// Return if no parameter is remaining...
IF ( ParameterCnt = 0 ) THEN RETURN; END_IF
// dec remaining parameter(s)                        
ParameterCnt := ParameterCnt - 1;
// Create log entry for OriginID
CreateLogMessagePara1 ( Timestamp   := Timestamp,
                        MessageType := MessageType.CMD,
                        Severity    := Severity.DEBUG,
                        MessageCode := 0,
                        MessageText := 'Response.OriginID = {1}',
                        Para1       :=  INT_TO_STRING(_response.OriginID));                       
                
END_METHOD

METHOD PROTECTED Reset : DINT
VAR_INPUT
END_VAR
                  Reset := SUPER^.Reset();

Done               := FALSE;
Busy               := FALSE;
ParameterAccepted  := FALSE;
CommandBuffered    := FALSE;
CommandAborted     := FALSE;
CommandInterrupted := FALSE;

                
END_METHOD
END_FUNCTION_BLOCK

/// Write default values of dynamic parameters used by move commands
FUNCTION_BLOCK MC_WriteRobotDefaultDynamicsFB EXTENDS RobotLibraryBaseExecuteFB
// ------------------------------------------------------------------------- 
//  SRCI Robot Library                                                
// ------------------------------------------------------------------------- 
//                                                                           
//  Object:      WriteRobotDefaultDynamicsFB                                       
//  Author:      Thorsten Brach                                                
//  Date:        2024-06-01
//
//  Description:                                              
//   
//                                                                           
//  Copyright: 
//    (C) 2024 Thorsten Brach. All rights reserved                                                                                                                                            
//             Licensed under the MIT License.
//                                                                           
//  Disclaimer:                                                                           
//    This project is provided without any guarantee and can be used for   
//    private and commercial purposes. Any use is at the user’s 
//    own risk and responsibility.
//
// -------------------------------------------------------------------------
VAR_INPUT
  /// command parameter 
  ParCmd             : WriteRobotDefaultDynamicsParCmd;
END_VAR
VAR_OUTPUT
  /// Command is transferred and confirmed by the RC
  CommandBuffered    : BOOL;
  /// The command was aborted by another command
  CommandAborted     : BOOL;
  /// TRUE, while command is interrupted during execution and can be continued.
  CommandInterrupted : BOOL;
  /// command outputs
  OutCmd             : WriteRobotDefaultDynamicsOutCmd;       
END_VAR

VAR
  /// internal copy of command parameter 
 _parCmd             : WriteRobotDefaultDynamicsParCmd;
  /// command data to send
 _command            : WriteRobotDefaultDynamicsSendData;
  /// response data received
 _response           : WriteRobotDefaultDynamicsRecvData;      
END_VAR

            SUPER^(AxesGroup := AxesGroup);
          

METHOD INTERNAL CheckAddParameter : BOOL
VAR_INPUT
  /// Payload pointer
  PayloadPtr : UDINT;
END_VAR
VAR
  /// Payload as byte array
  Payload    : ARRAY [1..SIZEOF(_command)] OF BYTE;
  /// Null Byte array 
  Null       : ARRAY [1..SIZEOF(_command)] OF BYTE;
  /// Data length to compare
  DataLen    : UDINT;
END_VAR
                  // Payload pointer must be decreased by one byte, because ADR(Payload) is already one byte !
PayloadPtr := LIMIT (0, PayloadPtr - 1, SIZEOF(Payload) -1);
// Convert command struct to payload array
SysDepMemCpy( pDest := ADR(Payload), pSrc := ADR(_command), DataLen := SIZEOF(_command));
// Calculate the data length to compare - at least one byte must be compared !
DataLen := LIMIT(1, SIZEOF(Payload) - PayloadPtr, SIZEOF(Payload)); 
// Compare Payload-Array with Null-Byte-Array
CheckAddParameter := SysDepMemCmp( pData1 := ADR(Payload) + PayloadPtr , pData2 := ADR(Null), DataLen := DataLen) <>  RobotLibraryConstants.OK ;
                
END_METHOD

METHOD PROTECTED CheckFunctionSupported : BOOL
VAR_IN_OUT
  /// Robot assignment of function
  AxesGroup : AxesGroup; 
END_VAR
                  CheckFunctionSupported := AxesGroup.State.RobotData.RCSupportedFunctions.WriteRobotDefaultDynamics;

IF ( NOT CheckFunctionSupported )
THEN
  // call base implementation for set error and create log entry
  SUPER^.CheckFunctionSupported(AxesGroup := AxesGroup);
END_IF
                
END_METHOD

METHOD PROTECTED CheckParameterChanged : BOOL
VAR_IN_OUT
  /// Robot assignment of function
  AxesGroup    : AxesGroup; 
END_VAR
                  // Check ParCmd Size is > 0, because MemCmp does not work correctly with size = 0
IF (SIZEOF(ParCmd) = 0) OR (_stepCmd = 0)
THEN 
  RETURN;
END_IF

// compare memory 
_parameterChanged := ( SysDepMemCmp(pData1 := ADR(ParCmd), pData2 := ADR(_parCmd), DataLen := SIZEOF(ParCmd)) <> RobotLibraryConstants.OK );

// check parameter valid ?
_parameterValid   := CheckParameterValid( AxesGroup := AxesGroup );

IF ((  _parameterChanged        )  AND 
    (  _parameterValid          )) OR
    (  _parameterUpdateInternal )  
THEN  
  // Create log entry for parameter changed event
  CreateLogMessagePara1 ( Timestamp   := AxesGroup.State.SystemTime,
                          MessageType := MessageType.CMD,
                          Severity    := Severity.DEBUG,
                          MessageCode := 0,
                          MessageText := 'NotifyParameterChanged Event {1}',
                          Para1       :=  '' );

  // reset internal flag for send parameter update
 _parameterUpdateInternal := FALSE;
  // update internal copy of parameters 
 _parCmd := ParCmd;
  // inc parameter sequence
 _command.ParSeq := _command.ParSeq + 1;
  // update command data  
  CommandData := CreateCommandPayload(AxesGroup := AxesGroup); // ( Access via reference to rCommandFB in ACR )
  // notify active command register 
  AxesGroup.Acyclic.ActiveCommandRegister.NotifyParameterChanged := _uniqueID;
END_IF
                
END_METHOD

METHOD PROTECTED CheckParameterValid : BOOL
VAR_IN_OUT
  /// Robot assignment of function
  AxesGroup : AxesGroup; 
END_VAR
VAR
  /// internal index for loops
 _idx : DINT;
END_VAR
                  CheckParameterValid := TRUE;


// Check ParCmd.DynamicValues.VelocityRate ? 
IF ( SysDepIsValidReal(ParCmd.DynamicValues.VelocityRate) = FALSE ) 
THEN
  // Parameter not valid
  CheckParameterValid := FALSE;
  // Set error
  SetError( ErrorID := RobotLibraryErrorIdEnum.ERR_VELOCITY_INVALID, Overwrite := TRUE );
  
  // Create log entry
  CreateLogMessagePara1 ( Timestamp   := AxesGroup.State.SystemTime,
                          MessageType := MessageType.CMD,
                          Severity    := Severity.ERROR,
                          MessageCode := ErrorID,
                          MessageText := 'Invalid Parameter ParCmd.DynamicValues.VelocityRate = {1}',
                          Para1       := VALID_REAL_TO_STRING(ParCmd.DynamicValues.VelocityRate));

  RETURN;                          
END_IF


// Check ParCmd.DynamicValues.AccelerationRate ? 
IF ( SysDepIsValidReal(ParCmd.DynamicValues.AccelerationRate) = FALSE ) 
THEN
  // Parameter not valid
  CheckParameterValid := FALSE;
  // Set error
  SetError( ErrorID := RobotLibraryErrorIdEnum.ERR_ACCELERATION_INVALID, Overwrite := TRUE );
  
  // Create log entry
  CreateLogMessagePara1 ( Timestamp   := AxesGroup.State.SystemTime,
                          MessageType := MessageType.CMD,
                          Severity    := Severity.ERROR,
                          MessageCode := ErrorID,
                          MessageText := 'Invalid Parameter ParCmd.DynamicValues.AccelerationRate = {1}',
                          Para1       := VALID_REAL_TO_STRING(ParCmd.DynamicValues.AccelerationRate));

  RETURN;                          
END_IF


// Check ParCmd.DynamicValues.DecelerationRate ? 
IF ( SysDepIsValidReal(ParCmd.DynamicValues.DecelerationRate) = FALSE ) 
THEN
  // Parameter not valid
  CheckParameterValid := FALSE;
  // Set error
  SetError( ErrorID := RobotLibraryErrorIdEnum.ERR_DECELERATION_INVALID, Overwrite := TRUE );
  
  // Create log entry
  CreateLogMessagePara1 ( Timestamp   := AxesGroup.State.SystemTime,
                          MessageType := MessageType.CMD,
                          Severity    := Severity.ERROR,
                          MessageCode := ErrorID,
                          MessageText := 'Invalid Parameter ParCmd.DynamicValues.DecelerationRate = {1}',
                          Para1       := VALID_REAL_TO_STRING(ParCmd.DynamicValues.DecelerationRate));

  RETURN;                          
END_IF


// Check ParCmd.DynamicValues.JerkRate ? 
IF ( SysDepIsValidReal(ParCmd.DynamicValues.JerkRate) = FALSE ) 
THEN
  // Parameter not valid
  CheckParameterValid := FALSE;
  // Set error
  SetError( ErrorID := RobotLibraryErrorIdEnum.ERR_JERK_INVALID, Overwrite := TRUE );
  
  // Create log entry
  CreateLogMessagePara1 ( Timestamp   := AxesGroup.State.SystemTime,
                          MessageType := MessageType.CMD,
                          Severity    := Severity.ERROR,
                          MessageCode := ErrorID,
                          MessageText := 'Invalid Parameter ParCmd.DynamicValues.JerkRate = {1}',
                          Para1       := VALID_REAL_TO_STRING(ParCmd.DynamicValues.JerkRate));

  RETURN;                          
END_IF
                
END_METHOD

METHOD INTERNAL CreateCommandPayload : RobotLibraryCommandDataFB
VAR_IN_OUT
  /// Robot assignment of function
  AxesGroup : AxesGroup; 
END_VAR
VAR
  /// Parameter count
 _parameterCnt : DINT;
END_VAR
// Table 6-146: Sent CMD payload (PLC to RC) of "WriteRobotDefaultDynamics"
// --------------------------
// Header
// --------------------------
// Byte 00 : UINT  - Type HB     
// Byte 01 :       - Type LB    
// Byte 02 : USINT - Reserve | ExecutionMode
// Byte 03 : USINT - ParSeq  | Priority
// --------------------------
// Datablock
// --------------------------
// Byte 04 : DATE Date
// Byte 05 : 
// Byte 06 : TIME_OF_DAY Time
// Byte 07 : 
// Byte 08 : 
// Byte 09 : UINT VelocityRate
// Byte 10 : 
// Byte 11 : 
// Byte 12 : UINT AccelerationRate
// Byte 13 : 
// Byte 14 : 
// Byte 15 : UINT DecelerationRate
// Byte 16 : 
// Byte 17 : 
// Byte 18 : UINT JerkRate
// --------------------------
                  // set command parameter 
_command.CmdTyp           :=  CmdType.WriteRobotDefaultDynamics;
_command.ExecMode         :=  ExecMode;
_command.ParSeq           := _command.ParSeq;
_command.Priority         :=  Priority;
_command.Timestamp        := _parCmd.DynamicValues.Timestamp;
_command.VelocityRate     := REAL_TO_PERCENT_UINT(_parCmd.DynamicValues.VelocityRate     , IsOptional := FALSE);
_command.AccelerationRate := REAL_TO_PERCENT_UINT(_parCmd.DynamicValues.AccelerationRate , IsOptional := FALSE);
_command.JerkRate         := REAL_TO_PERCENT_UINT(_parCmd.DynamicValues.JerkRate         , IsOptional := TRUE );
_command.DecelerationRate := REAL_TO_PERCENT_UINT(_parCmd.DynamicValues.DecelerationRate , IsOptional := TRUE );

// copy command data to header
_cmdHeader := _command;
// call base implementation to copy header to payload buffer
CreateCommandPayload := SUPER^.CreateCommandPayload(AxesGroup := AxesGroup);


// Check parameter must be added ? 
IF ( CheckAddParameter(CreateCommandPayload.PayloadPtr))
THEN
  // add command.DynamicValues.Timestamp.IEC_DATE
  CreateCommandPayload.AddUint(_command.Timestamp.IEC_DATE);
  // inc parameter counter
 _parameterCnt := _parameterCnt + 1;  
END_IF


// Check parameter must be added ? 
IF ( CheckAddParameter(CreateCommandPayload.PayloadPtr))
THEN
  // add command.DynamicValues.Timestamp.IEC_TIME
  CreateCommandPayload.AddTime(_command.Timestamp.IEC_TIME);
  // inc parameter counter
 _parameterCnt := _parameterCnt + 1;  
END_IF


// Check parameter must be added ? 
IF ( CheckAddParameter(CreateCommandPayload.PayloadPtr))
THEN
  // add command.DynamicValues.VelocityRate
  CreateCommandPayload.AddUint(_command.VelocityRate);
  // inc parameter counter
 _parameterCnt := _parameterCnt + 1;  
END_IF


// Check parameter must be added ? 
IF ( CheckAddParameter(CreateCommandPayload.PayloadPtr))
THEN
  // add command.DynamicValues.AccelerationRate
  CreateCommandPayload.AddUint(_command.AccelerationRate);
  // inc parameter counter
 _parameterCnt := _parameterCnt + 1;  
END_IF


// Check parameter must be added ? 
IF ( CheckAddParameter(CreateCommandPayload.PayloadPtr))
THEN
  // add command.DynamicValues.DecelerationRate
  CreateCommandPayload.AddUint(_command.DecelerationRate);
  // inc parameter counter
 _parameterCnt := _parameterCnt + 1;  
END_IF


// Check parameter must be added ? 
IF ( CheckAddParameter(CreateCommandPayload.PayloadPtr))
THEN
  // add command.DynamicValues.JerkRate
  CreateCommandPayload.AddUint(_command.JerkRate);
  // inc parameter counter
 _parameterCnt := _parameterCnt + 1;  
END_IF

 
// Create logging
CreateCommandPayloadLog(AxesGroup := AxesGroup, ParameterCnt := _parameterCnt);
                
END_METHOD

METHOD INTERNAL CreateCommandPayloadLog
VAR_IN_OUT
  /// Robot assignment of function
  AxesGroup : AxesGroup; 
END_VAR
VAR_INPUT
  /// Parameter count
  ParameterCnt : DINT;
END_VAR
                  // Create log entry for Parameter start
CreateLogMessagePara1 ( Timestamp   := AxesGroup.State.SystemTime,
                        MessageType := MessageType.CMD,
                        Severity    := Severity.DEBUG,
                        MessageCode := 0,
                        MessageText := 'Create command payload with {1} parameter(s) :',
                        Para1       := DINT_TO_STRING(ParameterCnt));
  

// Return if no parameter is remaining...
IF ( ParameterCnt = 0 ) THEN RETURN; END_IF
// dec remaining parameter(s)                        
ParameterCnt := ParameterCnt - 1;
// Create log entry for Timestamp.IEC_DATE
CreateLogMessagePara1 ( Timestamp   := AxesGroup.State.SystemTime,
                        MessageType := MessageType.CMD,
                        Severity    := Severity.DEBUG,
                        MessageCode := 0,
                        MessageText := 'Command.Timestamp.IEC_DATE = {1}',
                        Para1       :=  IEC_DATE_TO_STRING(_command.Timestamp.IEC_DATE));


// Return if no parameter is remaining...
IF ( ParameterCnt = 0 ) THEN RETURN; END_IF
// dec remaining parameter(s)                        
ParameterCnt := ParameterCnt - 1;
// Create log entry for Timestamp.IEC_TIME
CreateLogMessagePara1 ( Timestamp   := AxesGroup.State.SystemTime,
                        MessageType := MessageType.CMD,
                        Severity    := Severity.DEBUG,
                        MessageCode := 0,
                        MessageText := 'Command.Timestamp.IEC_TIME = {1}',
                        Para1       :=  IEC_TIME_TO_STRING(_command.Timestamp.IEC_TIME));


// Return if no parameter is remaining...
IF ( ParameterCnt = 0 ) THEN RETURN; END_IF
// dec remaining parameter(s)                        
ParameterCnt := ParameterCnt - 1;
// Create log entry for VelocityRate
CreateLogMessagePara1 ( Timestamp   := AxesGroup.State.SystemTime,
                        MessageType := MessageType.CMD,
                        Severity    := Severity.DEBUG,
                        MessageCode := 0,
                        MessageText := 'Command.VelocityRate = {1}',
                        Para1       :=  UINT_TO_STRING(_command.VelocityRate));


// Return if no parameter is remaining...
IF ( ParameterCnt = 0 ) THEN RETURN; END_IF
// dec remaining parameter(s)                        
ParameterCnt := ParameterCnt - 1;
// Create log entry for AccelerationRate
CreateLogMessagePara1 ( Timestamp   := AxesGroup.State.SystemTime,
                        MessageType := MessageType.CMD,
                        Severity    := Severity.DEBUG,
                        MessageCode := 0,
                        MessageText := 'Command.AccelerationRate = {1}',
                        Para1       :=  UINT_TO_STRING(_command.AccelerationRate));


// Return if no parameter is remaining...
IF ( ParameterCnt = 0 ) THEN RETURN; END_IF
// dec remaining parameter(s)                        
ParameterCnt := ParameterCnt - 1;
// Create log entry for DecelerationRate
CreateLogMessagePara1 ( Timestamp   := AxesGroup.State.SystemTime,
                        MessageType := MessageType.CMD,
                        Severity    := Severity.DEBUG,
                        MessageCode := 0,
                        MessageText := 'Command.DecelerationRate = {1}',
                        Para1       :=  UINT_TO_STRING(_command.DecelerationRate));


// Return if no parameter is remaining...
IF ( ParameterCnt = 0 ) THEN RETURN; END_IF
// dec remaining parameter(s)                        
ParameterCnt := ParameterCnt - 1;
// Create log entry for JerkRate
CreateLogMessagePara1 ( Timestamp   := AxesGroup.State.SystemTime,
                        MessageType := MessageType.CMD,
                        Severity    := Severity.DEBUG,
                        MessageCode := 0,
                        MessageText := 'Command.JerkRate = {1}',
                        Para1       :=  UINT_TO_STRING(_command.JerkRate));
                
END_METHOD

METHOD FB_init : BOOL
VAR_INPUT
  /// if TRUE, the retain variables are initialized (warm start / cold start)
  bInitRetains : BOOL; 
  /// if TRUE, the instance afterwards gets moved into the copy code (online change)
  bInCopyCode  : BOOL;  
END_VAR
                  MyType := 'MC_WriteRobotDefaultDynamicsFB';

ExecMode := ExecutionMode.PARALLEL;
Priority := PriorityLevel.NORMAL;
                
END_METHOD

METHOD PROTECTED OnApplyOutCmd
VAR_INPUT
  /// Command message state
  State : CmdMessageState;
END_VAR
                  IF ( State = CmdMessageState.EMPTY ) 
THEN
  // Reset command outputs
  SysDepMemSet(pDest := ADR(OutCmd), Value := 0, DataLen := SIZEOF(OutCmd));         
END_IF

IF (( State = CmdMessageState.ACTIVE ) OR
    ( State = CmdMessageState.DONE   ))
THEN
  // Update results
  OutCmd.DefaultDynamicValues.VelocityRate     := PERCENT_UINT_TO_REAL(_response.VelocityRate     , IsOptional := FALSE); 
  OutCmd.DefaultDynamicValues.AccelerationRate := PERCENT_UINT_TO_REAL(_response.AccelerationRate , IsOptional := FALSE);
  OutCmd.DefaultDynamicValues.DecelerationRate := PERCENT_UINT_TO_REAL(_response.DecelerationRate , IsOptional := TRUE );
  OutCmd.DefaultDynamicValues.JerkRate         := PERCENT_UINT_TO_REAL(_response.JerkRate         , IsOptional := TRUE );
END_IF
                
END_METHOD

METHOD PROTECTED OnExecRun : DINT
VAR_IN_OUT
  /// Robot assignment of function
  AxesGroup : AxesGroup; 
END_VAR
                  // call base implementation
SUPER^.OnExecRun(AxesGroup := AxesGroup);

CASE _stepCmd OF
  
  00:  IF ( _execute_R.Q ) AND ( NOT Error)  
       THEN
         // Check function is supported and parameter are valid ?
         IF (( CheckFunctionSupported( AxesGroup := AxesGroup )) AND
             ( CheckParameterValid   ( AxesGroup := AxesGroup )))
         THEN      
           // set busy flag
           Busy := TRUE;
           // Reset command outputs
           SysDepMemSet(pDest := ADR(OutCmd), Value := 0, DataLen := SIZEOF(OutCmd));         
           // apply command parameter
          _parCmd := ParCmd;
           // init parameter sequence
          _command.ParSeq := 1;
           // create command data
           CommandData := CreateCommandPayload(AxesGroup := AxesGroup);
           // Add command to active command register
          _uniqueID := AxesGroup.Acyclic.ActiveCommandRegister.AddCmd( pCommandFB := ADR(THIS^ ));     
           // set timeout
           SetTimeout(PT := _timeoutCmd, rTimer := _timerCmd);
           // inc step counter
          _stepCmd := _stepCmd + 1;
         END_IF 
       END_IF
     

  01:  // Wait for responce received
       IF ( _responseReceived )
       THEN
         // reset response received flag
        _responseReceived := FALSE;
         // update state flags
         OnUpdateStateFlags(_response.State);
         // update state flags
         OnApplyOutCmd(_response.State);

         // Done, Aborted or Error ?
         IF (_response.State >= CmdMessageState.DONE )
         THEN
           // Update the DefaultDynamics in user defined system datas 
           AxesGroup.SystemData.UpdateDefaultDynamics( DynamicValues := OutCmd.DefaultDynamicValues);
           // set timeout
           SetTimeout(PT := _timeoutCmd, rTimer := _timerCmd);
           // inc step counter
          _stepCmd := _stepCmd + 1; 
         END_IF
       END_IF


  02: IF ( NOT Execute)
      THEN
        Reset();  
      END_IF     

ELSE
  // invalid step
  SetError( ErrorID := RobotLibraryErrorIdEnum.ERR_INVALID_STEP, Overwrite := TRUE );
END_CASE


// Reset FB
IF ( NOT Execute )
THEN
  Reset();
END_IF
                
END_METHOD

METHOD PROTECTED OnUpdateStateFlags
VAR_INPUT
  /// Command message state
  State : CmdMessageState;
END_VAR
                  // Reset State flags
CommandInterrupted := FALSE;
CommandAborted     := FALSE;
Done               := FALSE;

CASE State OF

  // No operation or process is active
  CmdMessageState.EMPTY               :;
  // Created but not yet started
  CmdMessageState.CREATED             :;
  // Buffered and awaiting execution
  CmdMessageState.BUFFERED            : CommandBuffered   := TRUE;
  // Buffered in planner for future execution
  CmdMessageState.BUFFERED_IN_PLANNER : CommandBuffered   := TRUE;
  // Currently active and in progress
  CmdMessageState.ACTIVE              :;                                 
  // Interrupted and awaiting continuation
  CmdMessageState.INTERRUPTED         : CommandInterrupted := TRUE;     
  // Requested for abort
  CmdMessageState.ABORT_REQUEST       :;
  // Successfully completed
  CmdMessageState.DONE                : Done               := TRUE;
                                        Busy               := FALSE;
  // Aborted before completion
  CmdMessageState.ABORTED             : CommandAborted     := TRUE;
                                        Busy               := FALSE;
  // Encountered an error during execution
  CmdMessageState.ERROR               : Error              := TRUE;
                                        Busy               := FALSE;
END_CASE
                
END_METHOD

METHOD INTERNAL ParseResponsePayload : DINT
VAR_INPUT
  /// Response data
  ResponseData : RobotLibraryResponseDataFB;
  /// Timestamp
  Timestamp    : SystemTime;  
END_VAR
VAR
  /// Parameter count
 _parameterCnt : DINT;
END_VAR
// Table 6-147: Received CMD payload (RC to PLC) of "WriteRobotDefaultDynamics"
// --------------------------
// Header
// --------------------------
// Byte 00 : USINT   - ParSeq | State     
// Byte 01 : SINT    - AlarmMessageSeverity    
// Byte 02 : UINT    - AlarmMessageCode HB
// Byte 03 :         - AlarmMessageCode LB
// --------------------------
// Datablock
// --------------------------
// Byte 04 : UINT VelocityRate
// Byte 05 : 
// Byte 06 : UINT AccelerationRate
// Byte 07 : 
// Byte 08 : UINT DecelerationRate
// Byte 09 : 
// Byte 10 : UINT JerkRate
// Byte 11 : 
// --------------------------
                  // call base implementation to parse the header from payload buffer
ResponseData.PayloadPtr := SUPER^.ParseResponsePayload(ResponseData := ResponseData, Timestamp := Timestamp);

// copy parsed header to response
_response.ParSeq               := _rspHeader.ParSeq;
_response.State                := _rspHeader.State;
_response.AlarmMessageSeverity := _rspHeader.AlarmMessageSeverity;
_response.AlarmMessageCode     := _rspHeader.AlarmMessageCode;


// Check payload remaining ? 
IF ( ResponseData.IsPayloadRemaining)
THEN  
  // Get Response.VelocityRate
 _response.VelocityRate     := ResponseData.GetUint();
  // inc parameter counter
 _parameterCnt := _parameterCnt + 1;
END_IF


// Check payload remaining ? 
IF ( ResponseData.IsPayloadRemaining)
THEN  
  // Get Response.AccelerationRate
 _response.AccelerationRate := ResponseData.GetUint();
  // inc parameter counter
 _parameterCnt := _parameterCnt + 1;
END_IF


// Check payload remaining ? 
IF ( ResponseData.IsPayloadRemaining)
THEN  
  // Get Response.DecelerationRate
 _response.DecelerationRate := ResponseData.GetUint();
  // inc parameter counter
 _parameterCnt := _parameterCnt + 1;
END_IF


// Check payload remaining ? 
IF ( ResponseData.IsPayloadRemaining)
THEN  
  // Get Response.JerkRate
 _response.JerkRate         := ResponseData.GetUint();
  // inc parameter counter
 _parameterCnt := _parameterCnt + 1;
END_IF

 
// Create logging
ParseResponsePayloadLog(ResponseData := ResponseData, Timestamp := Timestamp, ParameterCnt := _parameterCnt);
                
END_METHOD

METHOD INTERNAL ParseResponsePayloadLog
VAR_INPUT
  /// Response data
  ResponseData : RobotLibraryResponseDataFB;
  /// Timestamp
  Timestamp    : SystemTime;  
  /// Parameter count
  ParameterCnt : DINT;
END_VAR
                  // Create log entry for Parameter start
CreateLogMessagePara1 ( Timestamp   := Timestamp,
                        MessageType := MessageType.CMD,
                        Severity    := Severity.DEBUG,
                        MessageCode := 0,
                        MessageText := '{1} parameter(s) to parse from the response data:',
                        Para1       := DINT_TO_STRING(ParameterCnt));
               

// Return if no parameter is remaining...
IF ( ParameterCnt = 0 ) THEN RETURN; END_IF
// dec remaining parameter(s)                        
ParameterCnt := ParameterCnt - 1;
// Create log entry for VelocityRate
CreateLogMessagePara1 ( Timestamp   := Timestamp,
                        MessageType := MessageType.CMD,
                        Severity    := Severity.DEBUG,
                        MessageCode := 0,
                        MessageText := 'Response.VelocityRate = {1}',
                        Para1       :=  UINT_TO_STRING(_response.VelocityRate));


// Return if no parameter is remaining...
IF ( ParameterCnt = 0 ) THEN RETURN; END_IF
// dec remaining parameter(s)                        
ParameterCnt := ParameterCnt - 1;
// Create log entry for AccelerationRate
CreateLogMessagePara1 ( Timestamp   := Timestamp,
                        MessageType := MessageType.CMD,
                        Severity    := Severity.DEBUG,
                        MessageCode := 0,
                        MessageText := 'Response.AccelerationRate = {1}',
                        Para1       :=  UINT_TO_STRING(_response.AccelerationRate));


// Return if no parameter is remaining...
IF ( ParameterCnt = 0 ) THEN RETURN; END_IF
// dec remaining parameter(s)                        
ParameterCnt := ParameterCnt - 1;
// Create log entry for DecelerationRate
CreateLogMessagePara1 ( Timestamp   := Timestamp,
                        MessageType := MessageType.CMD,
                        Severity    := Severity.DEBUG,
                        MessageCode := 0,
                        MessageText := 'Response.DecelerationRate = {1}',
                        Para1       :=  UINT_TO_STRING(_response.DecelerationRate));


// Return if no parameter is remaining...
IF ( ParameterCnt = 0 ) THEN RETURN; END_IF
// dec remaining parameter(s)                        
ParameterCnt := ParameterCnt - 1;
// Create log entry for JerkRate
CreateLogMessagePara1 ( Timestamp   := Timestamp,
                        MessageType := MessageType.CMD,
                        Severity    := Severity.DEBUG,
                        MessageCode := 0,
                        MessageText := 'Response.JerkRate = {1}',
                        Para1       :=  UINT_TO_STRING(_response.JerkRate));
                
END_METHOD

METHOD PROTECTED Reset : DINT
VAR_INPUT
END_VAR
                  Reset := SUPER^.Reset();

Done               := FALSE;
Busy               := FALSE;
CommandBuffered    := FALSE;
CommandAborted     := FALSE;
CommandInterrupted := FALSE;

                
END_METHOD
END_FUNCTION_BLOCK

/// Write reference values of robot dynamics for path movement
FUNCTION_BLOCK MC_WriteRobotReferenceDynamicsFB EXTENDS RobotLibraryBaseExecuteFB
// ------------------------------------------------------------------------- 
//  SRCI Robot Library                                                
// ------------------------------------------------------------------------- 
//                                                                           
//  Object:      WriteRobotReferenceDynamicsFB                                       
//  Author:      Thorsten Brach                                                
//  Date:        2024-06-01
//
//  Description:                                              
//   
//                                                                           
//  Copyright: 
//    (C) 2024 Thorsten Brach. All rights reserved                                                                                                                                            
//             Licensed under the MIT License.
//                                                                           
//  Disclaimer:                                                                           
//    This project is provided without any guarantee and can be used for   
//    private and commercial purposes. Any use is at the user’s 
//    own risk and responsibility.
//
// -------------------------------------------------------------------------
VAR_INPUT
  /// internal copy of command parameter 
  ParCmd             : WriteRobotReferenceDynamicsParCmd; 
END_VAR
VAR_OUTPUT
  /// Command is transferred and confirmed by the RC
  CommandBuffered    : BOOL;
  /// The command was aborted by another command
  CommandAborted     : BOOL;
  /// TRUE, while command is interrupted during execution and can be continued.
  CommandInterrupted : BOOL;
  /// command outputs
  OutCmd             : WriteRobotReferenceDynamicsOutCmd;       
END_VAR

VAR
  /// internal copy of command parameter 
 _parCmd             : WriteRobotReferenceDynamicsParCmd;
  /// command data to send
 _command            : WriteRobotReferenceDynamicsSendData;
  /// response data received
 _response           : WriteRobotReferenceDynamicsRecvData;      
END_VAR

            SUPER^(AxesGroup := AxesGroup);
          

METHOD INTERNAL CheckAddParameter : BOOL
VAR_INPUT
  /// Payload pointer
  PayloadPtr : UDINT;
END_VAR
VAR
  /// Payload as byte array
  Payload    : ARRAY [1..SIZEOF(_command)] OF BYTE;
  /// Null Byte array 
  Null       : ARRAY [1..SIZEOF(_command)] OF BYTE;
  /// Data length to compare
  DataLen    : UDINT;
END_VAR
                  // Payload pointer must be decreased by one byte, because ADR(Payload) is already one byte !
PayloadPtr := LIMIT (0, PayloadPtr - 1, SIZEOF(Payload) -1);
// Convert command struct to payload array
SysDepMemCpy( pDest := ADR(Payload), pSrc := ADR(_command), DataLen := SIZEOF(_command));
// Calculate the data length to compare - at least one byte must be compared !
DataLen := LIMIT(1, SIZEOF(Payload) - PayloadPtr, SIZEOF(Payload)); 
// Compare Payload-Array with Null-Byte-Array
CheckAddParameter := SysDepMemCmp( pData1 := ADR(Payload) + PayloadPtr , pData2 := ADR(Null), DataLen := DataLen) <>  RobotLibraryConstants.OK ;
                
END_METHOD

METHOD PROTECTED CheckFunctionSupported : BOOL
VAR_IN_OUT
  /// Robot assignment of function
  AxesGroup : AxesGroup; 
END_VAR
                  CheckFunctionSupported := AxesGroup.State.RobotData.RCSupportedFunctions.WriteRobotReferenceDynamics;

IF ( NOT CheckFunctionSupported )
THEN
  // call base implementation for set error and create log entry
  SUPER^.CheckFunctionSupported(AxesGroup := AxesGroup);
END_IF
                
END_METHOD

METHOD PROTECTED CheckParameterChanged : BOOL
VAR_IN_OUT
  /// Robot assignment of function
  AxesGroup    : AxesGroup; 
END_VAR
                  // Check ParCmd Size is > 0, because MemCmp does not work correctly with size = 0
IF (SIZEOF(ParCmd) = 0) OR (_stepCmd = 0)
THEN 
  RETURN;
END_IF

// compare memory 
_parameterChanged := ( SysDepMemCmp(pData1 := ADR(ParCmd), pData2 := ADR(_parCmd), DataLen := SIZEOF(ParCmd)) <> RobotLibraryConstants.OK );

// check parameter valid ?
_parameterValid   := CheckParameterValid( AxesGroup := AxesGroup );

IF ((  _parameterChanged        )  AND 
    (  _parameterValid          )) OR
    (  _parameterUpdateInternal )  
THEN  
  // Create log entry for parameter changed event
  CreateLogMessagePara1 ( Timestamp   := AxesGroup.State.SystemTime,
                          MessageType := MessageType.CMD,
                          Severity    := Severity.DEBUG,
                          MessageCode := 0,
                          MessageText := 'NotifyParameterChanged Event {1}',
                          Para1       :=  '' );

  // reset internal flag for send parameter update
 _parameterUpdateInternal := FALSE;
  // update internal copy of parameters 
 _parCmd := ParCmd;
  // inc parameter sequence
 _command.ParSeq := _command.ParSeq + 1;
  // update command data  
  CommandData := CreateCommandPayload(AxesGroup := AxesGroup); // ( Access via reference to rCommandFB in ACR )
  // notify active command register 
  AxesGroup.Acyclic.ActiveCommandRegister.NotifyParameterChanged := _uniqueID;
END_IF
                
END_METHOD

METHOD PROTECTED CheckParameterValid : BOOL
VAR_IN_OUT
  /// Robot assignment of function
  AxesGroup : AxesGroup; 
END_VAR
VAR
  /// internal index for loops
 _idx : DINT;
END_VAR
                  CheckParameterValid := TRUE;


// Check ParCmd.DynamicValues.VelocityReference ? 
IF ( SysDepIsValidReal(ParCmd.DynamicValues.VelocityReference) = FALSE ) 
THEN
  // Parameter not valid
  CheckParameterValid := FALSE;
  // Set error
  SetError( ErrorID := RobotLibraryErrorIdEnum.ERR_VELOCITY_INVALID, Overwrite := TRUE );
  
  // Create log entry
  CreateLogMessagePara1 ( Timestamp   := AxesGroup.State.SystemTime,
                          MessageType := MessageType.CMD,
                          Severity    := Severity.ERROR,
                          MessageCode := ErrorID,
                          MessageText := 'Invalid Parameter ParCmd.DynamicValues.VelocityReference = {1}',
                          Para1       := VALID_REAL_TO_STRING(ParCmd.DynamicValues.VelocityReference));

  RETURN;                          
END_IF


// Check ParCmd.DynamicValues.AccelerationReference ? 
IF ( SysDepIsValidReal(ParCmd.DynamicValues.AccelerationReference) = FALSE ) 
THEN
  // Parameter not valid
  CheckParameterValid := FALSE;
  // Set error
  SetError( ErrorID := RobotLibraryErrorIdEnum.ERR_ACCELERATION_INVALID, Overwrite := TRUE );
  
  // Create log entry
  CreateLogMessagePara1 ( Timestamp   := AxesGroup.State.SystemTime,
                          MessageType := MessageType.CMD,
                          Severity    := Severity.ERROR,
                          MessageCode := ErrorID,
                          MessageText := 'Invalid Parameter ParCmd.DynamicValues.AccelerationReference = {1}',
                          Para1       := VALID_REAL_TO_STRING(ParCmd.DynamicValues.AccelerationReference));

  RETURN;                          
END_IF


// Check ParCmd.DynamicValues.DecelerationReference ? 
IF ( SysDepIsValidReal(ParCmd.DynamicValues.DecelerationReference) = FALSE ) 
THEN
  // Parameter not valid
  CheckParameterValid := FALSE;
  // Set error
  SetError( ErrorID := RobotLibraryErrorIdEnum.ERR_DECELERATION_INVALID, Overwrite := TRUE );
  
  // Create log entry
  CreateLogMessagePara1 ( Timestamp   := AxesGroup.State.SystemTime,
                          MessageType := MessageType.CMD,
                          Severity    := Severity.ERROR,
                          MessageCode := ErrorID,
                          MessageText := 'Invalid Parameter ParCmd.DynamicValues.DecelerationReference = {1}',
                          Para1       := VALID_REAL_TO_STRING(ParCmd.DynamicValues.DecelerationReference));

  RETURN;                          
END_IF


// Check ParCmd.DynamicValues.JerkReference ? 
IF ( SysDepIsValidReal(ParCmd.DynamicValues.JerkReference) = FALSE ) 
THEN
  // Parameter not valid
  CheckParameterValid := FALSE;
  // Set error
  SetError( ErrorID := RobotLibraryErrorIdEnum.ERR_JERK_INVALID, Overwrite := TRUE );
  
  // Create log entry
  CreateLogMessagePara1 ( Timestamp   := AxesGroup.State.SystemTime,
                          MessageType := MessageType.CMD,
                          Severity    := Severity.ERROR,
                          MessageCode := ErrorID,
                          MessageText := 'Invalid Parameter ParCmd.DynamicValues.JerkReference = {1}',
                          Para1       := VALID_REAL_TO_STRING(ParCmd.DynamicValues.JerkReference));

  RETURN;                          
END_IF
                
END_METHOD

METHOD INTERNAL CreateCommandPayload : RobotLibraryCommandDataFB
VAR_IN_OUT
  /// Robot assignment of function
  AxesGroup : AxesGroup; 
END_VAR
VAR
  /// Parameter count
 _parameterCnt : DINT;
END_VAR
// Table 6-139: Sent CMD payload (PLC to RC) of "WriteRobotReferenceDynamics"
// --------------------------
// Header
// --------------------------
// Byte 00 : UINT  - Type HB     
// Byte 01 :       - Type LB    
// Byte 02 : USINT - Reserve | ExecutionMode
// Byte 03 : USINT - ParSeq  | Priority
// --------------------------
// Datablock
// --------------------------
// Byte 04 : DATE Date
// Byte 05 : 
// Byte 06 : TIME_OF_DAY Time
// Byte 07 : 
// Byte 08 : 
// Byte 09 : REAL VelocityReference
// Byte 10 : 
// Byte 11 : 
// Byte 12 : REAL AccelerationReference
// Byte 13 : 
// Byte 14 : 
// Byte 15 : REAL DecelerationReference
// Byte 16 : 
// Byte 17 : 
// Byte 18 : REAL JerkReference
// Byte 19 : 
// Byte 20 : 
// Byte 21 : 
// Byte 22 : REAL 
// Byte 23 : 
// Byte 24 : 
// Byte 25 : 
// --------------------------
                  // set command parameter 
_command.CmdTyp                :=  CmdType.WriteRobotReferenceDynamics;
_command.ExecMode              :=  ExecMode;
_command.ParSeq                := _command.ParSeq;
_command.Priority              :=  Priority;

_command.DynamicValues         := _parCmd.DynamicValues; {warning 'ToDo: Check if this is a mistake in the SRCI specification ? '}

(*
 _command.Timestamp             := _parCmd.DynamicValues.Timestamp;
 _command.VelocityReference     := REAL_TO_PERCENT_UINT(_parCmd.DynamicValues.VelocityReference     , IsOptional := FALSE);
 _command.AccelerationReference := REAL_TO_PERCENT_UINT(_parCmd.DynamicValues.AccelerationReference , IsOptional := FALSE);
 _command.JerkReference         := REAL_TO_PERCENT_UINT(_parCmd.DynamicValues.JerkReference         , IsOptional := TRUE );
 _command.DecelerationReference := REAL_TO_PERCENT_UINT(_parCmd.DynamicValues.DecelerationReference , IsOptional := TRUE );
*)

// copy command data to header
_cmdHeader := _command;
// call base implementation to copy header to payload buffer
CreateCommandPayload := SUPER^.CreateCommandPayload(AxesGroup := AxesGroup);


// Check parameter must be added ? 
IF ( CheckAddParameter(CreateCommandPayload.PayloadPtr))
THEN
  // add command.DynamicValues.Timestamp.IEC_DATE
  CreateCommandPayload.AddUint(_command.DynamicValues.Timestamp.IEC_DATE);
  // inc parameter counter
 _parameterCnt := _parameterCnt + 1;  
END_IF


// Check parameter must be added ? 
IF ( CheckAddParameter(CreateCommandPayload.PayloadPtr))
THEN
  // add command.DynamicValues.Timestamp.IEC_TIME
  CreateCommandPayload.AddTime(_command.DynamicValues.Timestamp.IEC_TIME);
  // inc parameter counter
 _parameterCnt := _parameterCnt + 1;  
END_IF


// Check parameter must be added ? 
IF ( CheckAddParameter(CreateCommandPayload.PayloadPtr))
THEN
  // add command.DynamicValues.VelocityReference
  CreateCommandPayload.AddReal(_command.DynamicValues.VelocityReference);
  // inc parameter counter
 _parameterCnt := _parameterCnt + 1;  
END_IF


// Check parameter must be added ? 
IF ( CheckAddParameter(CreateCommandPayload.PayloadPtr))
THEN
  // add command.DynamicValues.AccelerationReference
  CreateCommandPayload.AddReal(_command.DynamicValues.AccelerationReference);
  // inc parameter counter
 _parameterCnt := _parameterCnt + 1;  
END_IF


// Check parameter must be added ? 
IF ( CheckAddParameter(CreateCommandPayload.PayloadPtr))
THEN
  // add command.DynamicValues.DecelerationRate
  CreateCommandPayload.AddReal(_command.DynamicValues.DecelerationReference);
  // inc parameter counter
 _parameterCnt := _parameterCnt + 1;  
END_IF


// Check parameter must be added ? 
IF ( CheckAddParameter(CreateCommandPayload.PayloadPtr))
THEN
  // add command.DynamicValues.JerkRate
  CreateCommandPayload.AddReal(_command.DynamicValues.JerkReference);
  // inc parameter counter
 _parameterCnt := _parameterCnt + 1;  
END_IF
  
  
// Create logging
CreateCommandPayloadLog(AxesGroup := AxesGroup, ParameterCnt := _parameterCnt);
                
END_METHOD

METHOD INTERNAL CreateCommandPayloadLog
VAR_IN_OUT
  /// Robot assignment of function
  AxesGroup : AxesGroup; 
END_VAR
VAR_INPUT
  /// Parameter count
  ParameterCnt : DINT;
END_VAR
                  // Create log entry for Parameter start
CreateLogMessagePara1 ( Timestamp   := AxesGroup.State.SystemTime,
                        MessageType := MessageType.CMD,
                        Severity    := Severity.DEBUG,
                        MessageCode := 0,
                        MessageText := 'Create command payload with {1} parameter(s) :',
                        Para1       := DINT_TO_STRING(ParameterCnt));
  

// Return if no parameter is remaining...
IF ( ParameterCnt = 0 ) THEN RETURN; END_IF
// dec remaining parameter(s)                        
ParameterCnt := ParameterCnt - 1;
// Create log entry for DynamicValues.Timestamp.IEC_DATE
CreateLogMessagePara1 ( Timestamp   := AxesGroup.State.SystemTime,
                        MessageType := MessageType.CMD,
                        Severity    := Severity.DEBUG,
                        MessageCode := 0,
                        MessageText := 'Command.DynamicValues.Timestamp.IEC_DATE = {1}',
                        Para1       :=  IEC_DATE_TO_STRING(_command.DynamicValues.Timestamp.IEC_DATE));


// Return if no parameter is remaining...
IF ( ParameterCnt = 0 ) THEN RETURN; END_IF
// dec remaining parameter(s)                        
ParameterCnt := ParameterCnt - 1;
// Create log entry for DynamicValues.Timestamp.IEC_TIME
CreateLogMessagePara1 ( Timestamp   := AxesGroup.State.SystemTime,
                        MessageType := MessageType.CMD,
                        Severity    := Severity.DEBUG,
                        MessageCode := 0,
                        MessageText := 'Command.DynamicValues.Timestamp.IEC_TIME = {1}',
                        Para1       :=  IEC_TIME_TO_STRING(_command.DynamicValues.Timestamp.IEC_TIME));


// Return if no parameter is remaining...
IF ( ParameterCnt = 0 ) THEN RETURN; END_IF
// dec remaining parameter(s)                        
ParameterCnt := ParameterCnt - 1;
// Create log entry for DynamicValues.VelocityReference
CreateLogMessagePara1 ( Timestamp   := AxesGroup.State.SystemTime,
                        MessageType := MessageType.CMD,
                        Severity    := Severity.DEBUG,
                        MessageCode := 0,
                        MessageText := 'Command..DynamicValues.VelocityReference = {1}',
                        Para1       :=  REAL_TO_STRING(_command.DynamicValues.VelocityReference));


// Return if no parameter is remaining...
IF ( ParameterCnt = 0 ) THEN RETURN; END_IF
// dec remaining parameter(s)                        
ParameterCnt := ParameterCnt - 1;
// Create log entry for DynamicValues.AccelerationReference
CreateLogMessagePara1 ( Timestamp   := AxesGroup.State.SystemTime,
                        MessageType := MessageType.CMD,
                        Severity    := Severity.DEBUG,
                        MessageCode := 0,
                        MessageText := 'Command.DynamicValues.AccelerationReference = {1}',
                        Para1       :=  REAL_TO_STRING(_command.DynamicValues.AccelerationReference));


// Return if no parameter is remaining...
IF ( ParameterCnt = 0 ) THEN RETURN; END_IF
// dec remaining parameter(s)                        
ParameterCnt := ParameterCnt - 1;
// Create log entry for DynamicValues.DecelerationReference
CreateLogMessagePara1 ( Timestamp   := AxesGroup.State.SystemTime,
                        MessageType := MessageType.CMD,
                        Severity    := Severity.DEBUG,
                        MessageCode := 0,
                        MessageText := 'Command.DynamicValues.DecelerationReference = {1}',
                        Para1       :=  REAL_TO_STRING(_command.DynamicValues.DecelerationReference));


// Return if no parameter is remaining...
IF ( ParameterCnt = 0 ) THEN RETURN; END_IF
// dec remaining parameter(s)                        
ParameterCnt := ParameterCnt - 1;
// Create log entry for DynamicValues.JerkReference
CreateLogMessagePara1 ( Timestamp   := AxesGroup.State.SystemTime,
                        MessageType := MessageType.CMD,
                        Severity    := Severity.DEBUG,
                        MessageCode := 0,
                        MessageText := 'Command.DynamicValues.JerkReference = {1}',
                        Para1       :=  REAL_TO_STRING(_command.DynamicValues.JerkReference));
                
END_METHOD

METHOD FB_init : BOOL
VAR_INPUT
  /// if TRUE, the retain variables are initialized (warm start / cold start)
  bInitRetains : BOOL; 
  /// if TRUE, the instance afterwards gets moved into the copy code (online change)
  bInCopyCode  : BOOL;  
END_VAR
                  MyType := 'MC_WriteRobotReferenceDynamicsFB';

ExecMode := ExecutionMode.PARALLEL;
Priority := PriorityLevel.NORMAL;
                
END_METHOD

METHOD PROTECTED OnApplyOutCmd
VAR_INPUT
  /// Command message state
  State : CmdMessageState;
END_VAR
                  IF ( State = CmdMessageState.EMPTY ) 
THEN
  // Reset command outputs
  SysDepMemSet(pDest := ADR(OutCmd), Value := 0, DataLen := SIZEOF(OutCmd));         
END_IF

IF (( State = CmdMessageState.ACTIVE ) OR
    ( State = CmdMessageState.DONE   ))
THEN
  // Update results
  Outcmd.ReferenceDynamicValues.Timestamp             := _response.ReferenceDynamicValues.Timestamp;
  OutCmd.ReferenceDynamicValues.VelocityReference     := _response.ReferenceDynamicValues.VelocityReference; 
  OutCmd.ReferenceDynamicValues.AccelerationReference := _response.ReferenceDynamicValues.AccelerationReference;
  OutCmd.ReferenceDynamicValues.DecelerationReference := _response.ReferenceDynamicValues.DecelerationReference;
  OutCmd.ReferenceDynamicValues.JerkReference         := _response.ReferenceDynamicValues.JerkReference;
END_IF
                
END_METHOD

METHOD PROTECTED OnExecRun : DINT
VAR_IN_OUT
  /// Robot assignment of function
  AxesGroup : AxesGroup; 
END_VAR
                  // call base implementation
SUPER^.OnExecRun(AxesGroup := AxesGroup);

CASE _stepCmd OF
  
  00:  IF ( _execute_R.Q ) AND ( NOT Error)  
       THEN
         // Check function is supported and parameter are valid ?
         IF (( CheckFunctionSupported( AxesGroup := AxesGroup )) AND
             ( CheckParameterValid   ( AxesGroup := AxesGroup )))
         THEN      
           // set busy flag
           Busy := TRUE;
           // Reset command outputs
           SysDepMemSet(pDest := ADR(OutCmd), Value := 0, DataLen := SIZEOF(OutCmd));         
           // apply command parameter
          _parCmd := ParCmd;
           // init parameter sequence
          _command.ParSeq := 1;
           // create command data
           CommandData := CreateCommandPayload(AxesGroup := AxesGroup);
           // Add command to active command register
          _uniqueID := AxesGroup.Acyclic.ActiveCommandRegister.AddCmd( pCommandFB := ADR(THIS^ ));     
           // set timeout
           SetTimeout(PT := _timeoutCmd, rTimer := _timerCmd);
           // inc step counter
          _stepCmd := _stepCmd + 1;
         END_IF 
       END_IF
     

  01:  // Wait for responce received
       IF ( _responseReceived )
       THEN
         // reset response received flag
        _responseReceived := FALSE;
         // update state flags
         OnUpdateStateFlags(_response.State);
         // update state flags
         OnApplyOutCmd(_response.State);
               
         // Done, Aborted or Error ?
         IF (_response.State >= CmdMessageState.DONE )
         THEN
           // Update the ReferenceDynamics in user defined system datas 
           AxesGroup.SystemData.UpdateReferenceDynamics( DynamicValues := OutCmd.ReferenceDynamicValues);
           // set timeout
           SetTimeout(PT := _timeoutCmd, rTimer := _timerCmd);
           // inc step counter
          _stepCmd := _stepCmd + 1; 
         END_IF
       END_IF


  02: IF ( NOT Execute)
      THEN
        Reset();
      END_IF     

ELSE
  // invalid step
  SetError( ErrorID := RobotLibraryErrorIdEnum.ERR_INVALID_STEP, Overwrite := TRUE );
END_CASE


// Reset FB
IF ( NOT Execute )
THEN
  Reset();
END_IF
                
END_METHOD

METHOD PROTECTED OnUpdateStateFlags
VAR_INPUT
  /// Command message state
  State : CmdMessageState;
END_VAR
                  // Reset State flags
CommandInterrupted := FALSE;
CommandAborted     := FALSE;
Done               := FALSE;

CASE State OF

  // No operation or process is active
  CmdMessageState.EMPTY               :;
  // Created but not yet started
  CmdMessageState.CREATED             :;
  // Buffered and awaiting execution
  CmdMessageState.BUFFERED            : CommandBuffered   := TRUE;
  // Buffered in planner for future execution
  CmdMessageState.BUFFERED_IN_PLANNER : CommandBuffered   := TRUE;
  // Currently active and in progress
  CmdMessageState.ACTIVE              :;                                 
  // Interrupted and awaiting continuation
  CmdMessageState.INTERRUPTED         : CommandInterrupted := TRUE;     
  // Requested for abort
  CmdMessageState.ABORT_REQUEST       :;
  // Successfully completed
  CmdMessageState.DONE                : Done               := TRUE;
                                        Busy               := FALSE;
  // Aborted before completion
  CmdMessageState.ABORTED             : CommandAborted     := TRUE;
                                        Busy               := FALSE;
  // Encountered an error during execution
  CmdMessageState.ERROR               : Error              := TRUE;
                                        Busy               := FALSE;
END_CASE
                
END_METHOD

METHOD INTERNAL ParseResponsePayload : DINT
VAR_INPUT
  /// Response data
  ResponseData : RobotLibraryResponseDataFB;
  /// Timestamp
  Timestamp    : SystemTime;  
END_VAR
VAR
  /// Parameter count
 _parameterCnt : DINT;
END_VAR
// Table 6-140: Received CMD payload (RC to PLC) of "WriteRobotReferenceDynamics"
// --------------------------
// Header
// --------------------------
// Byte 00 : USINT   - ParSeq | State     
// Byte 01 : SINT    - AlarmMessageSeverity    
// Byte 02 : UINT    - AlarmMessageCode HB
// Byte 03 :         - AlarmMessageCode LB
// --------------------------
// Datablock
// --------------------------
// Byte 04 : REAL VelocityReference
// Byte 05 : 
// Byte 06 : 
// Byte 07 : 
// Byte 08 : REAL AccelerationReference
// Byte 09 : 
// Byte 10 : 
// Byte 11 : 
// Byte 12 : REAL DecelerationReference
// Byte 13 : 
// Byte 14 : 
// Byte 15 : 
// Byte 16 : REAL JerkReference
// Byte 17 : 
// Byte 18 : 
// Byte 19 : 
// --------------------------
                  // call base implementation to parse the header from payload buffer
ResponseData.PayloadPtr := SUPER^.ParseResponsePayload(ResponseData := ResponseData, Timestamp := Timestamp);

// copy parsed header to response
_response.ParSeq               := _rspHeader.ParSeq;
_response.State                := _rspHeader.State;
_response.AlarmMessageSeverity := _rspHeader.AlarmMessageSeverity;
_response.AlarmMessageCode     := _rspHeader.AlarmMessageCode;


// Check payload remaining ? 
IF ( ResponseData.IsPayloadRemaining)
THEN  
  // Get Response.ReferenceDynamicValues.VelocityReference
 _response.ReferenceDynamicValues.VelocityReference := ResponseData.GetReal();
  // inc parameter counter
 _parameterCnt := _parameterCnt + 1;
END_IF


// Check payload remaining ? 
IF ( ResponseData.IsPayloadRemaining)
THEN  
  // Get Response.ReferenceDynamicValues.AccelerationReference
 _response.ReferenceDynamicValues.AccelerationReference := ResponseData.GetReal();
  // inc parameter counter
 _parameterCnt := _parameterCnt + 1;
END_IF


// Check payload remaining ? 
IF ( ResponseData.IsPayloadRemaining)
THEN  
  // Get Response.ReferenceDynamicValues.DecelerationReference
 _response.ReferenceDynamicValues.DecelerationReference := ResponseData.GetReal();
  // inc parameter counter
 _parameterCnt := _parameterCnt + 1;
END_IF


// Check payload remaining ? 
IF ( ResponseData.IsPayloadRemaining)
THEN  
  // Get ReferenceDynamicValues.JerkReference
 _response.ReferenceDynamicValues.JerkReference := ResponseData.GetReal();
  // inc parameter counter
 _parameterCnt := _parameterCnt + 1;
END_IF

 
// Create logging
ParseResponsePayloadLog(ResponseData := ResponseData, Timestamp := Timestamp, ParameterCnt := _parameterCnt);
                
END_METHOD

METHOD INTERNAL ParseResponsePayloadLog
VAR_INPUT
  /// Response data
  ResponseData : RobotLibraryResponseDataFB;
  /// Timestamp
  Timestamp    : SystemTime;  
  /// Parameter count
  ParameterCnt : DINT;
END_VAR
                  // Create log entry for Parameter start
CreateLogMessagePara1 ( Timestamp   := Timestamp,
                        MessageType := MessageType.CMD,
                        Severity    := Severity.DEBUG,
                        MessageCode := 0,
                        MessageText := '{1} parameter(s) to parse from the response data:',
                        Para1       := DINT_TO_STRING(ParameterCnt));


// Return if no parameter is remaining...
IF ( ParameterCnt = 0 ) THEN RETURN; END_IF
// dec remaining parameter(s)                        
ParameterCnt := ParameterCnt - 1;
// Create log entry for ReferenceDynamicValues.VelocityReference
CreateLogMessagePara1 ( Timestamp   := Timestamp,
                        MessageType := MessageType.CMD,
                        Severity    := Severity.DEBUG,
                        MessageCode := 0,
                        MessageText := 'Response.ReferenceDynamicValues.VelocityReference = {1}',
                        Para1       :=  REAL_TO_STRING(_response.ReferenceDynamicValues.VelocityReference));


// Return if no parameter is remaining...
IF ( ParameterCnt = 0 ) THEN RETURN; END_IF
// dec remaining parameter(s)                        
ParameterCnt := ParameterCnt - 1;
// Create log entry for ReferenceDynamicValues.AccelerationReference
CreateLogMessagePara1 ( Timestamp   := Timestamp,
                        MessageType := MessageType.CMD,
                        Severity    := Severity.DEBUG,
                        MessageCode := 0,
                        MessageText := 'Response.ReferenceDynamicValues.AccelerationReference = {1}',
                        Para1       :=  REAL_TO_STRING(_response.ReferenceDynamicValues.AccelerationReference));
                        

// Return if no parameter is remaining...
IF ( ParameterCnt = 0 ) THEN RETURN; END_IF
// dec remaining parameter(s)                        
ParameterCnt := ParameterCnt - 1;
// Create log entry for ReferenceDynamicValues.DecelerationReference
CreateLogMessagePara1 ( Timestamp   := Timestamp,
                        MessageType := MessageType.CMD,
                        Severity    := Severity.DEBUG,
                        MessageCode := 0,
                        MessageText := 'Response.ReferenceDynamicValues.DecelerationReference = {1}',
                        Para1       :=  REAL_TO_STRING(_response.ReferenceDynamicValues.DecelerationReference));


// Return if no parameter is remaining...
IF ( ParameterCnt = 0 ) THEN RETURN; END_IF
// dec remaining parameter(s)                        
ParameterCnt := ParameterCnt - 1;
// Create log entry for ReferenceDynamicValues.JerkReference
CreateLogMessagePara1 ( Timestamp   := Timestamp,
                        MessageType := MessageType.CMD,
                        Severity    := Severity.DEBUG,
                        MessageCode := 0,
                        MessageText := 'Response.ReferenceDynamicValues.JerkReference = {1}',
                        Para1       :=  REAL_TO_STRING(_response.ReferenceDynamicValues.JerkReference));
                
END_METHOD

METHOD PROTECTED Reset : DINT
VAR_INPUT
END_VAR
                  Reset := SUPER^.Reset();

Done               := FALSE;
Busy               := FALSE;
CommandBuffered    := FALSE;
CommandAborted     := FALSE;
CommandInterrupted := FALSE;

                
END_METHOD
END_FUNCTION_BLOCK

/// Change robot limits of robot axes (degree)
FUNCTION_BLOCK MC_WriteRobotSWLimitsFB EXTENDS RobotLibraryBaseExecuteFB
// ------------------------------------------------------------------------- 
//  SRCI Robot Library                                                
// ------------------------------------------------------------------------- 
//                                                                           
//  Object:      WriteRobotSWLimitsFB                                       
//  Author:      Thorsten Brach                                                
//  Date:        2024-06-01
//
//  Description:                                              
//   
//                                                                           
//  Copyright: 
//    (C) 2024 Thorsten Brach. All rights reserved                                                                                                                                            
//             Licensed under the MIT License.
//                                                                           
//  Disclaimer:                                                                           
//    This project is provided without any guarantee and can be used for   
//    private and commercial purposes. Any use is at the user’s 
//    own risk and responsibility.
//
// -------------------------------------------------------------------------
VAR_INPUT
  /// command parameter 
  ParCmd          : WriteRobotSWLimitsParCmd;
END_VAR
VAR_OUTPUT
  /// Command is transferred and confirmed by the RC
  CommandBuffered : BOOL;
  /// command outputs
  OutCmd          : WriteRobotSWLimitsOutCmd;       
END_VAR

VAR
  /// internal copy of command parameter 
 _parCmd          : WriteRobotSWLimitsParCmd;
  /// command data to send
 _command         : WriteRobotSWLimitsSendData;
  /// response data received
 _response        : WriteRobotSWLimitsRecvData;      
END_VAR

            SUPER^(AxesGroup := AxesGroup);
          

METHOD INTERNAL CheckAddParameter : BOOL
VAR_INPUT
  /// Payload pointer
  PayloadPtr : UDINT;
END_VAR
VAR
  /// Payload as byte array
  Payload    : ARRAY [1..SIZEOF(_command)] OF BYTE;
  /// Null Byte array 
  Null       : ARRAY [1..SIZEOF(_command)] OF BYTE;
  /// Data length to compare
  DataLen    : UDINT;
END_VAR
                  // Payload pointer must be decreased by one byte, because ADR(Payload) is already one byte !
PayloadPtr := LIMIT (0, PayloadPtr - 1, SIZEOF(Payload) -1);
// Convert command struct to payload array
SysDepMemCpy( pDest := ADR(Payload), pSrc := ADR(_command), DataLen := SIZEOF(_command));
// Calculate the data length to compare - at least one byte must be compared !
DataLen := LIMIT(1, SIZEOF(Payload) - PayloadPtr, SIZEOF(Payload)); 
// Compare Payload-Array with Null-Byte-Array
CheckAddParameter := SysDepMemCmp( pData1 := ADR(Payload) + PayloadPtr , pData2 := ADR(Null), DataLen := DataLen) <>  RobotLibraryConstants.OK ;
                
END_METHOD

METHOD PROTECTED CheckFunctionSupported : BOOL
VAR_IN_OUT
  /// Robot assignment of function
  AxesGroup : AxesGroup; 
END_VAR
                  CheckFunctionSupported := AxesGroup.State.RobotData.RCSupportedFunctions.WriteRobotSWLimits;

IF ( NOT CheckFunctionSupported )
THEN
  // call base implementation for set error and create log entry
  SUPER^.CheckFunctionSupported(AxesGroup := AxesGroup);
END_IF
                
END_METHOD

METHOD PROTECTED CheckParameterChanged : BOOL
VAR_IN_OUT
  /// Robot assignment of function
  AxesGroup    : AxesGroup; 
END_VAR
                  // Check ParCmd Size is > 0, because MemCmp does not work correctly with size = 0
IF (SIZEOF(ParCmd) = 0) OR (_stepCmd = 0)
THEN 
  RETURN;
END_IF

// compare memory 
_parameterChanged := ( SysDepMemCmp(pData1 := ADR(ParCmd), pData2 := ADR(_parCmd), DataLen := SIZEOF(ParCmd)) <> RobotLibraryConstants.OK );

// check parameter valid ?
_parameterValid   := CheckParameterValid( AxesGroup := AxesGroup );

IF ((  _parameterChanged        )  AND 
    (  _parameterValid          )) OR
    (  _parameterUpdateInternal )  
THEN  
  // Create log entry for parameter changed event
  CreateLogMessagePara1 ( Timestamp   := AxesGroup.State.SystemTime,
                          MessageType := MessageType.CMD,
                          Severity    := Severity.DEBUG,
                          MessageCode := 0,
                          MessageText := 'NotifyParameterChanged Event {1}',
                          Para1       :=  '' );

  // reset internal flag for send parameter update
 _parameterUpdateInternal := FALSE;
  // update internal copy of parameters 
 _parCmd := ParCmd;
  // inc parameter sequence
 _command.ParSeq := _command.ParSeq + 1;
  // update command data  
  CommandData := CreateCommandPayload(AxesGroup := AxesGroup); // ( Access via reference to rCommandFB in ACR )
  // notify active command register 
  AxesGroup.Acyclic.ActiveCommandRegister.NotifyParameterChanged := _uniqueID;
END_IF
                
END_METHOD

METHOD PROTECTED CheckParameterValid : BOOL
VAR_IN_OUT
  /// Robot assignment of function
  AxesGroup : AxesGroup; 
END_VAR
VAR
  /// internal index for loops
 _idx : DINT;
END_VAR
                  CheckParameterValid := TRUE;


// Check ParCmd.LimitValues.J1LowerLimit ? 
IF ( SysDepIsValidReal(ParCmd.LimitValues.J1LowerLimit) = FALSE ) 
THEN
  // Parameter not valid
  CheckParameterValid := FALSE;
  // Set error
  SetError( ErrorID := RobotLibraryErrorIdEnum.ERR_INVALID_PAR_CMD, Overwrite := TRUE );
  
  // Create log entry
  CreateLogMessagePara1 ( Timestamp   := AxesGroup.State.SystemTime,
                          MessageType := MessageType.CMD,
                          Severity    := Severity.ERROR,
                          MessageCode := ErrorID,
                          MessageText := 'Invalid Parameter ParCmd.LimitValues.J1LowerLimit = {1}',
                          Para1       := VALID_REAL_TO_STRING(ParCmd.LimitValues.J1LowerLimit));

  RETURN;                          
END_IF


// Check ParCmd.LimitValues.J1UpperLimit ? 
IF ( SysDepIsValidReal(ParCmd.LimitValues.J1UpperLimit) = FALSE ) 
THEN
  // Parameter not valid
  CheckParameterValid := FALSE;
  // Set error
  SetError( ErrorID := RobotLibraryErrorIdEnum.ERR_INVALID_PAR_CMD, Overwrite := TRUE );
  
  // Create log entry
  CreateLogMessagePara1 ( Timestamp   := AxesGroup.State.SystemTime,
                          MessageType := MessageType.CMD,
                          Severity    := Severity.ERROR,
                          MessageCode := ErrorID,
                          MessageText := 'Invalid Parameter ParCmd.LimitValues.J1UpperLimit = {1}',
                          Para1       := VALID_REAL_TO_STRING(ParCmd.LimitValues.J1UpperLimit));

  RETURN;                          
END_IF


// Check ParCmd.LimitValues.J2LowerLimit ? 
IF ( SysDepIsValidReal(ParCmd.LimitValues.J2LowerLimit) = FALSE ) 
THEN
  // Parameter not valid
  CheckParameterValid := FALSE;
  // Set error
  SetError( ErrorID := RobotLibraryErrorIdEnum.ERR_INVALID_PAR_CMD, Overwrite := TRUE );
  
  // Create log entry
  CreateLogMessagePara1 ( Timestamp   := AxesGroup.State.SystemTime,
                          MessageType := MessageType.CMD,
                          Severity    := Severity.ERROR,
                          MessageCode := ErrorID,
                          MessageText := 'Invalid Parameter ParCmd.LimitValues.J2LowerLimit = {1}',
                          Para1       := VALID_REAL_TO_STRING(ParCmd.LimitValues.J2LowerLimit));

  RETURN;                          
END_IF


// Check ParCmd.LimitValues.J2UpperLimit ? 
IF ( SysDepIsValidReal(ParCmd.LimitValues.J2UpperLimit) = FALSE ) 
THEN
  // Parameter not valid
  CheckParameterValid := FALSE;
  // Set error
  SetError( ErrorID := RobotLibraryErrorIdEnum.ERR_INVALID_PAR_CMD, Overwrite := TRUE );
  
  // Create log entry
  CreateLogMessagePara1 ( Timestamp   := AxesGroup.State.SystemTime,
                          MessageType := MessageType.CMD,
                          Severity    := Severity.ERROR,
                          MessageCode := ErrorID,
                          MessageText := 'Invalid Parameter ParCmd.LimitValues.J2UpperLimit = {1}',
                          Para1       := VALID_REAL_TO_STRING(ParCmd.LimitValues.J2UpperLimit));

  RETURN;                          
END_IF


// Check ParCmd.LimitValues.J3LowerLimit ? 
IF ( SysDepIsValidReal(ParCmd.LimitValues.J3LowerLimit) = FALSE ) 
THEN
  // Parameter not valid
  CheckParameterValid := FALSE;
  // Set error
  SetError( ErrorID := RobotLibraryErrorIdEnum.ERR_INVALID_PAR_CMD, Overwrite := TRUE );
  
  // Create log entry
  CreateLogMessagePara1 ( Timestamp   := AxesGroup.State.SystemTime,
                          MessageType := MessageType.CMD,
                          Severity    := Severity.ERROR,
                          MessageCode := ErrorID,
                          MessageText := 'Invalid Parameter ParCmd.LimitValues.J3LowerLimit = {1}',
                          Para1       := VALID_REAL_TO_STRING(ParCmd.LimitValues.J3LowerLimit));

  RETURN;                          
END_IF


// Check ParCmd.LimitValues.J3UpperLimit ? 
IF ( SysDepIsValidReal(ParCmd.LimitValues.J3UpperLimit) = FALSE ) 
THEN
  // Parameter not valid
  CheckParameterValid := FALSE;
  // Set error
  SetError( ErrorID := RobotLibraryErrorIdEnum.ERR_INVALID_PAR_CMD, Overwrite := TRUE );
  
  // Create log entry
  CreateLogMessagePara1 ( Timestamp   := AxesGroup.State.SystemTime,
                          MessageType := MessageType.CMD,
                          Severity    := Severity.ERROR,
                          MessageCode := ErrorID,
                          MessageText := 'Invalid Parameter ParCmd.LimitValues.J3UpperLimit = {1}',
                          Para1       := VALID_REAL_TO_STRING(ParCmd.LimitValues.J3UpperLimit));

  RETURN;                          
END_IF


// Check ParCmd.LimitValues.J4LowerLimit ? 
IF ( SysDepIsValidReal(ParCmd.LimitValues.J4LowerLimit) = FALSE ) 
THEN
  // Parameter not valid
  CheckParameterValid := FALSE;
  // Set error
  SetError( ErrorID := RobotLibraryErrorIdEnum.ERR_INVALID_PAR_CMD, Overwrite := TRUE );
  
  // Create log entry
  CreateLogMessagePara1 ( Timestamp   := AxesGroup.State.SystemTime,
                          MessageType := MessageType.CMD,
                          Severity    := Severity.ERROR,
                          MessageCode := ErrorID,
                          MessageText := 'Invalid Parameter ParCmd.LimitValues.J4LowerLimit = {1}',
                          Para1       := VALID_REAL_TO_STRING(ParCmd.LimitValues.J4LowerLimit));

  RETURN;                          
END_IF


// Check ParCmd.LimitValues.J4UpperLimit ? 
IF ( SysDepIsValidReal(ParCmd.LimitValues.J4UpperLimit) = FALSE ) 
THEN
  // Parameter not valid
  CheckParameterValid := FALSE;
  // Set error
  SetError( ErrorID := RobotLibraryErrorIdEnum.ERR_INVALID_PAR_CMD, Overwrite := TRUE );
  
  // Create log entry
  CreateLogMessagePara1 ( Timestamp   := AxesGroup.State.SystemTime,
                          MessageType := MessageType.CMD,
                          Severity    := Severity.ERROR,
                          MessageCode := ErrorID,
                          MessageText := 'Invalid Parameter ParCmd.LimitValues.J4UpperLimit = {1}',
                          Para1       := VALID_REAL_TO_STRING(ParCmd.LimitValues.J4UpperLimit));

  RETURN;                          
END_IF


// Check ParCmd.LimitValues.J5LowerLimit ? 
IF ( SysDepIsValidReal(ParCmd.LimitValues.J5LowerLimit) = FALSE ) 
THEN
  // Parameter not valid
  CheckParameterValid := FALSE;
  // Set error
  SetError( ErrorID := RobotLibraryErrorIdEnum.ERR_INVALID_PAR_CMD, Overwrite := TRUE );
  
  // Create log entry
  CreateLogMessagePara1 ( Timestamp   := AxesGroup.State.SystemTime,
                          MessageType := MessageType.CMD,
                          Severity    := Severity.ERROR,
                          MessageCode := ErrorID,
                          MessageText := 'Invalid Parameter ParCmd.LimitValues.J5LowerLimit = {1}',
                          Para1       := VALID_REAL_TO_STRING(ParCmd.LimitValues.J5LowerLimit));

  RETURN;                          
END_IF


// Check ParCmd.LimitValues.J5UpperLimit ? 
IF ( SysDepIsValidReal(ParCmd.LimitValues.J5UpperLimit) = FALSE ) 
THEN
  // Parameter not valid
  CheckParameterValid := FALSE;
  // Set error
  SetError( ErrorID := RobotLibraryErrorIdEnum.ERR_INVALID_PAR_CMD, Overwrite := TRUE );
  
  // Create log entry
  CreateLogMessagePara1 ( Timestamp   := AxesGroup.State.SystemTime,
                          MessageType := MessageType.CMD,
                          Severity    := Severity.ERROR,
                          MessageCode := ErrorID,
                          MessageText := 'Invalid Parameter ParCmd.LimitValues.J5UpperLimit = {1}',
                          Para1       := VALID_REAL_TO_STRING(ParCmd.LimitValues.J5UpperLimit));

  RETURN;                          
END_IF


// Check ParCmd.LimitValues.J6LowerLimit ? 
IF ( SysDepIsValidReal(ParCmd.LimitValues.J6LowerLimit) = FALSE ) 
THEN
  // Parameter not valid
  CheckParameterValid := FALSE;
  // Set error
  SetError( ErrorID := RobotLibraryErrorIdEnum.ERR_INVALID_PAR_CMD, Overwrite := TRUE );
  
  // Create log entry
  CreateLogMessagePara1 ( Timestamp   := AxesGroup.State.SystemTime,
                          MessageType := MessageType.CMD,
                          Severity    := Severity.ERROR,
                          MessageCode := ErrorID,
                          MessageText := 'Invalid Parameter ParCmd.LimitValues.J6LowerLimit = {1}',
                          Para1       := VALID_REAL_TO_STRING(ParCmd.LimitValues.J6LowerLimit));

  RETURN;                          
END_IF


// Check ParCmd.LimitValues.J6UpperLimit ? 
IF ( SysDepIsValidReal(ParCmd.LimitValues.J6UpperLimit) = FALSE ) 
THEN
  // Parameter not valid
  CheckParameterValid := FALSE;
  // Set error
  SetError( ErrorID := RobotLibraryErrorIdEnum.ERR_INVALID_PAR_CMD, Overwrite := TRUE );
  
  // Create log entry
  CreateLogMessagePara1 ( Timestamp   := AxesGroup.State.SystemTime,
                          MessageType := MessageType.CMD,
                          Severity    := Severity.ERROR,
                          MessageCode := ErrorID,
                          MessageText := 'Invalid Parameter ParCmd.LimitValues.J6UpperLimit = {1}',
                          Para1       := VALID_REAL_TO_STRING(ParCmd.LimitValues.J6UpperLimit));

  RETURN;                          
END_IF


// Check ParCmd.LimitValues.E1LowerLimit ? 
IF ( SysDepIsValidReal(ParCmd.LimitValues.E1LowerLimit) = FALSE ) 
THEN
  // Parameter not valid
  CheckParameterValid := FALSE;
  // Set error
  SetError( ErrorID := RobotLibraryErrorIdEnum.ERR_INVALID_PAR_CMD, Overwrite := TRUE );
  
  // Create log entry
  CreateLogMessagePara1 ( Timestamp   := AxesGroup.State.SystemTime,
                          MessageType := MessageType.CMD,
                          Severity    := Severity.ERROR,
                          MessageCode := ErrorID,
                          MessageText := 'Invalid Parameter ParCmd.LimitValues.E1LowerLimit = {1}',
                          Para1       := VALID_REAL_TO_STRING(ParCmd.LimitValues.E1LowerLimit));

  RETURN;                          
END_IF


// Check ParCmd.LimitValues.E1UpperLimit ? 
IF ( SysDepIsValidReal(ParCmd.LimitValues.E1UpperLimit) = FALSE ) 
THEN
  // Parameter not valid
  CheckParameterValid := FALSE;
  // Set error
  SetError( ErrorID := RobotLibraryErrorIdEnum.ERR_INVALID_PAR_CMD, Overwrite := TRUE );
  
  // Create log entry
  CreateLogMessagePara1 ( Timestamp   := AxesGroup.State.SystemTime,
                          MessageType := MessageType.CMD,
                          Severity    := Severity.ERROR,
                          MessageCode := ErrorID,
                          MessageText := 'Invalid Parameter ParCmd.LimitValues.E1UpperLimit = {1}',
                          Para1       := VALID_REAL_TO_STRING(ParCmd.LimitValues.E1UpperLimit));

  RETURN;                          
END_IF


// Check ParCmd.LimitValues.E2LowerLimit ? 
IF ( SysDepIsValidReal(ParCmd.LimitValues.E2LowerLimit) = FALSE ) 
THEN
  // Parameter not valid
  CheckParameterValid := FALSE;
  // Set error
  SetError( ErrorID := RobotLibraryErrorIdEnum.ERR_INVALID_PAR_CMD, Overwrite := TRUE );
  
  // Create log entry
  CreateLogMessagePara1 ( Timestamp   := AxesGroup.State.SystemTime,
                          MessageType := MessageType.CMD,
                          Severity    := Severity.ERROR,
                          MessageCode := ErrorID,
                          MessageText := 'Invalid Parameter ParCmd.LimitValues.E2LowerLimit = {1}',
                          Para1       := VALID_REAL_TO_STRING(ParCmd.LimitValues.E2LowerLimit));

  RETURN;                          
END_IF


// Check ParCmd.LimitValues.E2UpperLimit ? 
IF ( SysDepIsValidReal(ParCmd.LimitValues.E2UpperLimit) = FALSE ) 
THEN
  // Parameter not valid
  CheckParameterValid := FALSE;
  // Set error
  SetError( ErrorID := RobotLibraryErrorIdEnum.ERR_INVALID_PAR_CMD, Overwrite := TRUE );
  
  // Create log entry
  CreateLogMessagePara1 ( Timestamp   := AxesGroup.State.SystemTime,
                          MessageType := MessageType.CMD,
                          Severity    := Severity.ERROR,
                          MessageCode := ErrorID,
                          MessageText := 'Invalid Parameter ParCmd.LimitValues.E2UpperLimit = {1}',
                          Para1       := VALID_REAL_TO_STRING(ParCmd.LimitValues.E2UpperLimit));

  RETURN;                          
END_IF


// Check ParCmd.LimitValues.E3LowerLimit ? 
IF ( SysDepIsValidReal(ParCmd.LimitValues.E3LowerLimit) = FALSE ) 
THEN
  // Parameter not valid
  CheckParameterValid := FALSE;
  // Set error
  SetError( ErrorID := RobotLibraryErrorIdEnum.ERR_INVALID_PAR_CMD, Overwrite := TRUE );
  
  // Create log entry
  CreateLogMessagePara1 ( Timestamp   := AxesGroup.State.SystemTime,
                          MessageType := MessageType.CMD,
                          Severity    := Severity.ERROR,
                          MessageCode := ErrorID,
                          MessageText := 'Invalid Parameter ParCmd.LimitValues.E3LowerLimit = {1}',
                          Para1       := VALID_REAL_TO_STRING(ParCmd.LimitValues.E3LowerLimit));

  RETURN;                          
END_IF


// Check ParCmd.LimitValues.E3UpperLimit ? 
IF ( SysDepIsValidReal(ParCmd.LimitValues.E3UpperLimit) = FALSE ) 
THEN
  // Parameter not valid
  CheckParameterValid := FALSE;
  // Set error
  SetError( ErrorID := RobotLibraryErrorIdEnum.ERR_INVALID_PAR_CMD, Overwrite := TRUE );
  
  // Create log entry
  CreateLogMessagePara1 ( Timestamp   := AxesGroup.State.SystemTime,
                          MessageType := MessageType.CMD,
                          Severity    := Severity.ERROR,
                          MessageCode := ErrorID,
                          MessageText := 'Invalid Parameter ParCmd.LimitValues.E3UpperLimit = {1}',
                          Para1       := VALID_REAL_TO_STRING(ParCmd.LimitValues.E3UpperLimit));

  RETURN;                          
END_IF


// Check ParCmd.LimitValues.E4LowerLimit ? 
IF ( SysDepIsValidReal(ParCmd.LimitValues.E4LowerLimit) = FALSE ) 
THEN
  // Parameter not valid
  CheckParameterValid := FALSE;
  // Set error
  SetError( ErrorID := RobotLibraryErrorIdEnum.ERR_INVALID_PAR_CMD, Overwrite := TRUE );
  
  // Create log entry
  CreateLogMessagePara1 ( Timestamp   := AxesGroup.State.SystemTime,
                          MessageType := MessageType.CMD,
                          Severity    := Severity.ERROR,
                          MessageCode := ErrorID,
                          MessageText := 'Invalid Parameter ParCmd.LimitValues.E4LowerLimit = {1}',
                          Para1       := VALID_REAL_TO_STRING(ParCmd.LimitValues.E4LowerLimit));

  RETURN;                          
END_IF


// Check ParCmd.LimitValues.E4UpperLimit ? 
IF ( SysDepIsValidReal(ParCmd.LimitValues.E4UpperLimit) = FALSE ) 
THEN
  // Parameter not valid
  CheckParameterValid := FALSE;
  // Set error
  SetError( ErrorID := RobotLibraryErrorIdEnum.ERR_INVALID_PAR_CMD, Overwrite := TRUE );
  
  // Create log entry
  CreateLogMessagePara1 ( Timestamp   := AxesGroup.State.SystemTime,
                          MessageType := MessageType.CMD,
                          Severity    := Severity.ERROR,
                          MessageCode := ErrorID,
                          MessageText := 'Invalid Parameter ParCmd.LimitValues.E4UpperLimit = {1}',
                          Para1       := VALID_REAL_TO_STRING(ParCmd.LimitValues.E4UpperLimit));

  RETURN;                          
END_IF


// Check ParCmd.LimitValues.E5LowerLimit ? 
IF ( SysDepIsValidReal(ParCmd.LimitValues.E5LowerLimit) = FALSE ) 
THEN
  // Parameter not valid
  CheckParameterValid := FALSE;
  // Set error
  SetError( ErrorID := RobotLibraryErrorIdEnum.ERR_INVALID_PAR_CMD, Overwrite := TRUE );
  
  // Create log entry
  CreateLogMessagePara1 ( Timestamp   := AxesGroup.State.SystemTime,
                          MessageType := MessageType.CMD,
                          Severity    := Severity.ERROR,
                          MessageCode := ErrorID,
                          MessageText := 'Invalid Parameter ParCmd.LimitValues.E5LowerLimit = {1}',
                          Para1       := VALID_REAL_TO_STRING(ParCmd.LimitValues.E5LowerLimit));

  RETURN;                          
END_IF


// Check ParCmd.LimitValues.E5UpperLimit ? 
IF ( SysDepIsValidReal(ParCmd.LimitValues.E5UpperLimit) = FALSE ) 
THEN
  // Parameter not valid
  CheckParameterValid := FALSE;
  // Set error
  SetError( ErrorID := RobotLibraryErrorIdEnum.ERR_INVALID_PAR_CMD, Overwrite := TRUE );
  
  // Create log entry
  CreateLogMessagePara1 ( Timestamp   := AxesGroup.State.SystemTime,
                          MessageType := MessageType.CMD,
                          Severity    := Severity.ERROR,
                          MessageCode := ErrorID,
                          MessageText := 'Invalid Parameter ParCmd.LimitValues.E5UpperLimit = {1}',
                          Para1       := VALID_REAL_TO_STRING(ParCmd.LimitValues.E5UpperLimit));

  RETURN;                          
END_IF


// Check ParCmd.LimitValues.E6LowerLimit ? 
IF ( SysDepIsValidReal(ParCmd.LimitValues.E6LowerLimit) = FALSE ) 
THEN
  // Parameter not valid
  CheckParameterValid := FALSE;
  // Set error
  SetError( ErrorID := RobotLibraryErrorIdEnum.ERR_INVALID_PAR_CMD, Overwrite := TRUE );
  
  // Create log entry
  CreateLogMessagePara1 ( Timestamp   := AxesGroup.State.SystemTime,
                          MessageType := MessageType.CMD,
                          Severity    := Severity.ERROR,
                          MessageCode := ErrorID,
                          MessageText := 'Invalid Parameter ParCmd.LimitValues.E6LowerLimit = {1}',
                          Para1       := VALID_REAL_TO_STRING(ParCmd.LimitValues.E6LowerLimit));

  RETURN;                          
END_IF


// Check ParCmd.LimitValues.E6UpperLimit ? 
IF ( SysDepIsValidReal(ParCmd.LimitValues.E6UpperLimit) = FALSE ) 
THEN
  // Parameter not valid
  CheckParameterValid := FALSE;
  // Set error
  SetError( ErrorID := RobotLibraryErrorIdEnum.ERR_INVALID_PAR_CMD, Overwrite := TRUE );
  
  // Create log entry
  CreateLogMessagePara1 ( Timestamp   := AxesGroup.State.SystemTime,
                          MessageType := MessageType.CMD,
                          Severity    := Severity.ERROR,
                          MessageCode := ErrorID,
                          MessageText := 'Invalid Parameter ParCmd.LimitValues.E6UpperLimit = {1}',
                          Para1       := VALID_REAL_TO_STRING(ParCmd.LimitValues.E6UpperLimit));

  RETURN;                          
END_IF


// Check ParCmd.ResetToFactoryDefaults ? 
IF (( ParCmd.ResetToFactoryDefaults <> FALSE ) AND
    ( ParCmd.ResetToFactoryDefaults <> TRUE  ))
THEN
  // Parameter not valid
  CheckParameterValid := FALSE;
  // Set error
  SetError( ErrorID := RobotLibraryErrorIdEnum.ERR_INVALID_PAR_CMD, Overwrite := TRUE );
  
  // Create log entry
  CreateLogMessagePara1 ( Timestamp   := AxesGroup.State.SystemTime,
                          MessageType := MessageType.CMD,
                          Severity    := Severity.ERROR,
                          MessageCode := ErrorID,
                          MessageText := 'Invalid Parameter ParCmd.ResetToFactoryDefaults = {1}',
                          Para1       := BOOL_TO_STRING(ParCmd.ResetToFactoryDefaults));

  RETURN;                          
END_IF
                
END_METHOD

METHOD INTERNAL CreateCommandPayload : RobotLibraryCommandDataFB
VAR_IN_OUT
  /// Robot assignment of function
  AxesGroup : AxesGroup; 
END_VAR
VAR
  /// Parameter count
 _parameterCnt : DINT;
END_VAR
// Table 6-185: Sent CMD payload (PLC to RC) of "WriteRobotSWLimits"
// --------------------------
// Header
// --------------------------
// Byte 00 : UINT  - Type HB     
// Byte 01 :       - Type LB    
// Byte 02 : USINT - Reserve | ExecutionMode
// Byte 03 : USINT - ParSeq  | Priority
// --------------------------
// Datablock
// --------------------------
// Byte 04 : DATE Date
// Byte 05 : 
// Byte 06 : TIME_OF_DAY Time
// Byte 07 : 
// Byte 08 : 
// Byte 09 : REAL J1LowerLimit
// Byte 10 : 
// Byte 11 : 
// Byte 12 : REAL J2LowerLimit
// Byte 13 : 
// Byte 14 : 
// Byte 15 : REAL J3LowerLimit
// Byte 16 : 
// Byte 17 : 
// Byte 18 : REAL J4LowerLimit
// Byte 19 : 
// Byte 20 : 
// Byte 21 : REAL J5LowerLimit
// Byte 22 : 
// Byte 23 : 
// Byte 24 : REAL J6LowerLimit
// Byte 25 : 
// Byte 26 : 
// Byte 27 : REAL E1LowerLimit
// Byte 28 : 
// Byte 29 : 
// Byte 30 : REAL J1UpperLimit
// Byte 31 : 
// Byte 32 : 
// Byte 33 : REAL J2UpperLimit
// Byte 34 : 
// Byte 35 : 
// Byte 36 : REAL J3UpperLimit
// Byte 37 : 
// Byte 38 : 
// Byte 39 : REAL J4UpperLimit
// Byte 40 : 
// Byte 41 : 
// Byte 42 : REAL J5UpperLimit
// Byte 43 : 
// Byte 44 : 
// Byte 45 : REAL J6UpperLimit
// Byte 46 : 
// Byte 47 : 
// Byte 48 : REAL E1UpperLimit
// Byte 49 : 
// Byte 50 : 
// Byte 51 : REAL E2LowerLimit
// Byte 52 : 
// Byte 53 : 
// Byte 54 : REAL E3LowerLimit
// Byte 55 : 
// Byte 56 : 
// Byte 57 : REAL E4LowerLimit
// Byte 58 : 
// Byte 59 : 
// Byte 60 : REAL E5LowerLimit
// Byte 61 : 
// Byte 62 : 
// Byte 63 : REAL E6LowerLimit
// Byte 64 : 
// Byte 65 : 
// Byte 66 : REAL E2UpperLimit
// Byte 67 : 
// Byte 68 : 
// Byte 69 : REAL E3UpperLimit
// Byte 70 : 
// Byte 71 : 
// Byte 72 : REAL E4UpperLimit
// Byte 73 : 
// Byte 74 : 
// Byte 75 : REAL E5UpperLimit
// Byte 76 : 
// Byte 77 : 
// Byte 78 : REAL E6UpperLimit
// Byte 79 : 
// Byte 80 : 
// Byte 81 : 
// Byte 82 : BOOL ResetToFactoryDefault
// --------------------------
                  // set command parameter 
_command.CmdTyp                 :=  CmdType.WriteRobotSWLimits;
_command.ExecMode               :=  ExecMode;
_command.ParSeq                 := _command.ParSeq;
_command.Priority               :=  Priority;
                                
_command.LimitValues            :=  _parCmd.LimitValues;
_command.ResetToFactoryDefaults :=  _parCmd.ResetToFactoryDefaults;

// copy command data to header
_cmdHeader := _command;
// call base implementation to copy header to payload buffer
CreateCommandPayload := SUPER^.CreateCommandPayload(AxesGroup := AxesGroup);


// Check parameter must be added ? 
IF ( CheckAddParameter(CreateCommandPayload.PayloadPtr))
THEN
  // add command.LimitValues.Timestamp.IEC_DATE
  CreateCommandPayload.AddUint(_command.LimitValues.Timestamp.IEC_DATE);
  // inc parameter counter
 _parameterCnt := _parameterCnt + 1;  
END_IF


// Check parameter must be added ? 
IF ( CheckAddParameter(CreateCommandPayload.PayloadPtr))
THEN
  // add command.LimitValues.Timestamp.IEC_TIME
  CreateCommandPayload.AddTime(_command.LimitValues.Timestamp.IEC_TIME);
  // inc parameter counter
 _parameterCnt := _parameterCnt + 1;  
END_IF


// Check parameter must be added ? 
IF ( CheckAddParameter(CreateCommandPayload.PayloadPtr))
THEN
  // add command.LimitValues.J1LowerLimit
  CreateCommandPayload.AddReal(_command.LimitValues.J1LowerLimit);
  // inc parameter counter
 _parameterCnt := _parameterCnt + 1;  
END_IF


// Check parameter must be added ? 
IF ( CheckAddParameter(CreateCommandPayload.PayloadPtr))
THEN
  // add command.LimitValues.J2LowerLimit
  CreateCommandPayload.AddReal(_command.LimitValues.J2LowerLimit);
  // inc parameter counter
 _parameterCnt := _parameterCnt + 1;  
END_IF


// Check parameter must be added ? 
IF ( CheckAddParameter(CreateCommandPayload.PayloadPtr))
THEN
  // add command.LimitValues.J3LowerLimit
  CreateCommandPayload.AddReal(_command.LimitValues.J3LowerLimit);
  // inc parameter counter
 _parameterCnt := _parameterCnt + 1;  
END_IF


// Check parameter must be added ? 
IF ( CheckAddParameter(CreateCommandPayload.PayloadPtr))
THEN
  // add command.LimitValues.J41LowerLimit
  CreateCommandPayload.AddReal(_command.LimitValues.J4LowerLimit);
  // inc parameter counter
 _parameterCnt := _parameterCnt + 1;  
END_IF


// Check parameter must be added ? 
IF ( CheckAddParameter(CreateCommandPayload.PayloadPtr))
THEN
  // add command.LimitValues.J5LowerLimit
  CreateCommandPayload.AddReal(_command.LimitValues.J5LowerLimit);
  // inc parameter counter
 _parameterCnt := _parameterCnt + 1;  
END_IF


// Check parameter must be added ? 
IF ( CheckAddParameter(CreateCommandPayload.PayloadPtr))
THEN
  // add command.LimitValues.J6LowerLimit
  CreateCommandPayload.AddReal(_command.LimitValues.J6LowerLimit);
  // inc parameter counter
 _parameterCnt := _parameterCnt + 1;  
END_IF


// Check parameter must be added ? 
IF ( CheckAddParameter(CreateCommandPayload.PayloadPtr))
THEN
  // add command.LimitValues.E1LowerLimit
  CreateCommandPayload.AddReal(_command.LimitValues.E1LowerLimit);
  // inc parameter counter
 _parameterCnt := _parameterCnt + 1;  
END_IF


// Check parameter must be added ? 
IF ( CheckAddParameter(CreateCommandPayload.PayloadPtr))
THEN
  // add command.LimitValues.J1UpperLimit
  CreateCommandPayload.AddReal(_command.LimitValues.J1UpperLimit);
  // inc parameter counter
 _parameterCnt := _parameterCnt + 1;  
END_IF


// Check parameter must be added ? 
IF ( CheckAddParameter(CreateCommandPayload.PayloadPtr))
THEN
  // add command.LimitValues.J2UpperLimit
  CreateCommandPayload.AddReal(_command.LimitValues.J2UpperLimit);
  // inc parameter counter
 _parameterCnt := _parameterCnt + 1;  
END_IF


// Check parameter must be added ? 
IF ( CheckAddParameter(CreateCommandPayload.PayloadPtr))
THEN
  // add command.LimitValues.J3UpperLimit
  CreateCommandPayload.AddReal(_command.LimitValues.J3UpperLimit);
  // inc parameter counter
 _parameterCnt := _parameterCnt + 1;  
END_IF


// Check parameter must be added ? 
IF ( CheckAddParameter(CreateCommandPayload.PayloadPtr))
THEN
  // add command.LimitValues.J4UpperLimit
  CreateCommandPayload.AddReal(_command.LimitValues.J4UpperLimit);
  // inc parameter counter
 _parameterCnt := _parameterCnt + 1;  
END_IF


// Check parameter must be added ? 
IF ( CheckAddParameter(CreateCommandPayload.PayloadPtr))
THEN
  // add command.LimitValues.J5UpperLimit
  CreateCommandPayload.AddReal(_command.LimitValues.J5UpperLimit);
  // inc parameter counter
 _parameterCnt := _parameterCnt + 1;  
END_IF


// Check parameter must be added ? 
IF ( CheckAddParameter(CreateCommandPayload.PayloadPtr))
THEN
  // add command.LimitValues.J6UpperLimit
  CreateCommandPayload.AddReal(_command.LimitValues.J6UpperLimit);
  // inc parameter counter
 _parameterCnt := _parameterCnt + 1;  
END_IF


// Check parameter must be added ? 
IF ( CheckAddParameter(CreateCommandPayload.PayloadPtr))
THEN
  // add command.LimitValues.E1UpperLimit
  CreateCommandPayload.AddReal(_command.LimitValues.E1UpperLimit);
  // inc parameter counter
 _parameterCnt := _parameterCnt + 1;  
END_IF


// Check parameter must be added ? 
IF ( CheckAddParameter(CreateCommandPayload.PayloadPtr))
THEN
  // add command.LimitValues.E2LowerLimit
  CreateCommandPayload.AddReal(_command.LimitValues.E2LowerLimit);
  // inc parameter counter
 _parameterCnt := _parameterCnt + 1;  
END_IF


// Check parameter must be added ? 
IF ( CheckAddParameter(CreateCommandPayload.PayloadPtr))
THEN
  // add command.LimitValues.E3LowerLimit
  CreateCommandPayload.AddReal(_command.LimitValues.E3LowerLimit);
  // inc parameter counter
 _parameterCnt := _parameterCnt + 1;  
END_IF


// Check parameter must be added ? 
IF ( CheckAddParameter(CreateCommandPayload.PayloadPtr))
THEN
  // add command.LimitValues.E4LowerLimit
  CreateCommandPayload.AddReal(_command.LimitValues.E4LowerLimit);
  // inc parameter counter
 _parameterCnt := _parameterCnt + 1;  
END_IF


// Check parameter must be added ? 
IF ( CheckAddParameter(CreateCommandPayload.PayloadPtr))
THEN
  // add command.LimitValues.E5LowerLimit
  CreateCommandPayload.AddReal(_command.LimitValues.E5LowerLimit);
  // inc parameter counter
 _parameterCnt := _parameterCnt + 1;  
END_IF


// Check parameter must be added ? 
IF ( CheckAddParameter(CreateCommandPayload.PayloadPtr))
THEN
  // add command.LimitValues.E6LowerLimit
  CreateCommandPayload.AddReal(_command.LimitValues.E6LowerLimit);
  // inc parameter counter
 _parameterCnt := _parameterCnt + 1;  
END_IF


// Check parameter must be added ? 
IF ( CheckAddParameter(CreateCommandPayload.PayloadPtr))
THEN
  // add command.LimitValues.E2UpperLimit
  CreateCommandPayload.AddReal(_command.LimitValues.E2UpperLimit);
  // inc parameter counter
 _parameterCnt := _parameterCnt + 1;  
END_IF


// Check parameter must be added ? 
IF ( CheckAddParameter(CreateCommandPayload.PayloadPtr))
THEN
  // add command.LimitValues.E3UpperLimit
  CreateCommandPayload.AddReal(_command.LimitValues.E3UpperLimit);
  // inc parameter counter
 _parameterCnt := _parameterCnt + 1;  
END_IF


// Check parameter must be added ? 
IF ( CheckAddParameter(CreateCommandPayload.PayloadPtr))
THEN
  // add command.LimitValues.E4UpperLimit
  CreateCommandPayload.AddReal(_command.LimitValues.E4UpperLimit);
  // inc parameter counter
 _parameterCnt := _parameterCnt + 1;  
END_IF


// Check parameter must be added ? 
IF ( CheckAddParameter(CreateCommandPayload.PayloadPtr))
THEN
  // add command.LimitValues.E5UpperLimit
  CreateCommandPayload.AddReal(_command.LimitValues.E5UpperLimit);
  // inc parameter counter
 _parameterCnt := _parameterCnt + 1;  
END_IF


// Check parameter must be added ? 
IF ( CheckAddParameter(CreateCommandPayload.PayloadPtr))
THEN
  // add command.LimitValues.E6UpperLimit
  CreateCommandPayload.AddReal(_command.LimitValues.E6UpperLimit);
  // inc parameter counter
 _parameterCnt := _parameterCnt + 1;  
END_IF

  
// Create logging
CreateCommandPayloadLog(AxesGroup := AxesGroup, ParameterCnt := _parameterCnt);
                
END_METHOD

METHOD INTERNAL CreateCommandPayloadLog
VAR_IN_OUT
  /// Robot assignment of function
  AxesGroup : AxesGroup; 
END_VAR
VAR_INPUT
  /// Parameter count
  ParameterCnt : DINT;
END_VAR
                  // Create log entry for Parameter start
CreateLogMessagePara1 ( Timestamp   := AxesGroup.State.SystemTime,
                        MessageType := MessageType.CMD,
                        Severity    := Severity.DEBUG,
                        MessageCode := 0,
                        MessageText := 'Create command payload with {1} parameter(s) :',
                        Para1       := DINT_TO_STRING(ParameterCnt));
  

// Return if no parameter is remaining...
IF ( ParameterCnt = 0 ) THEN RETURN; END_IF
// dec remaining parameter(s)                        
ParameterCnt := ParameterCnt - 1;
// Create log entry for LimitValues.Timestamp.IEC_DATE
CreateLogMessagePara1 ( Timestamp   := AxesGroup.State.SystemTime,
                        MessageType := MessageType.CMD,
                        Severity    := Severity.DEBUG,
                        MessageCode := 0,
                        MessageText := 'Command.LimitValues.Timestamp.IEC_DATE = {1}',
                        Para1       :=  IEC_DATE_TO_STRING(_command.LimitValues.Timestamp.IEC_DATE));


// Return if no parameter is remaining...
IF ( ParameterCnt = 0 ) THEN RETURN; END_IF
// dec remaining parameter(s)                        
ParameterCnt := ParameterCnt - 1;
// Create log entry for LimitValues.Timestamp.IEC_TIME
CreateLogMessagePara1 ( Timestamp   := AxesGroup.State.SystemTime,
                        MessageType := MessageType.CMD,
                        Severity    := Severity.DEBUG,
                        MessageCode := 0,
                        MessageText := 'Command.LimitValues.Timestamp.IEC_TIME = {1}',
                        Para1       :=  IEC_TIME_TO_STRING(_command.LimitValues.Timestamp.IEC_TIME));


// Return if no parameter is remaining...
IF ( ParameterCnt = 0 ) THEN RETURN; END_IF
// dec remaining parameter(s)                        
ParameterCnt := ParameterCnt - 1;
// Create log entry for LimitValues.J1LowerLimit
CreateLogMessagePara1 ( Timestamp   := AxesGroup.State.SystemTime,
                        MessageType := MessageType.CMD,
                        Severity    := Severity.DEBUG,
                        MessageCode := 0,
                        MessageText := 'Command.LimitValues.J1LowerLimit = {1}',
                        Para1       :=  REAL_TO_STRING(_command.LimitValues.J1LowerLimit));


// Return if no parameter is remaining...
IF ( ParameterCnt = 0 ) THEN RETURN; END_IF
// dec remaining parameter(s)                        
ParameterCnt := ParameterCnt - 1;
// Create log entry for LimitValues.J2LowerLimit
CreateLogMessagePara1 ( Timestamp   := AxesGroup.State.SystemTime,
                        MessageType := MessageType.CMD,
                        Severity    := Severity.DEBUG,
                        MessageCode := 0,
                        MessageText := 'Command.LimitValues.J2LowerLimit = {1}',
                        Para1       :=  REAL_TO_STRING(_command.LimitValues.J2LowerLimit));
                        

// Return if no parameter is remaining...
IF ( ParameterCnt = 0 ) THEN RETURN; END_IF
// dec remaining parameter(s)                        
ParameterCnt := ParameterCnt - 1;
// Create log entry for LimitValues.J3LowerLimit
CreateLogMessagePara1 ( Timestamp   := AxesGroup.State.SystemTime,
                        MessageType := MessageType.CMD,
                        Severity    := Severity.DEBUG,
                        MessageCode := 0,
                        MessageText := 'Command.LimitValues.J3LowerLimit = {1}',
                        Para1       :=  REAL_TO_STRING(_command.LimitValues.J3LowerLimit));
                        

// Return if no parameter is remaining...
IF ( ParameterCnt = 0 ) THEN RETURN; END_IF
// dec remaining parameter(s)                        
ParameterCnt := ParameterCnt - 1;
// Create log entry for LimitValues.J4LowerLimit
CreateLogMessagePara1 ( Timestamp   := AxesGroup.State.SystemTime,
                        MessageType := MessageType.CMD,
                        Severity    := Severity.DEBUG,
                        MessageCode := 0,
                        MessageText := 'Command.LimitValues.J4LowerLimit = {1}',
                        Para1       :=  REAL_TO_STRING(_command.LimitValues.J4LowerLimit));


// Return if no parameter is remaining...
IF ( ParameterCnt = 0 ) THEN RETURN; END_IF
// dec remaining parameter(s)                        
ParameterCnt := ParameterCnt - 1;
// Create log entry for LimitValues.J5LowerLimit
CreateLogMessagePara1 ( Timestamp   := AxesGroup.State.SystemTime,
                        MessageType := MessageType.CMD,
                        Severity    := Severity.DEBUG,
                        MessageCode := 0,
                        MessageText := 'Command.LimitValues.J5LowerLimit = {1}',
                        Para1       :=  REAL_TO_STRING(_command.LimitValues.J5LowerLimit));


// Return if no parameter is remaining...
IF ( ParameterCnt = 0 ) THEN RETURN; END_IF
// dec remaining parameter(s)                        
ParameterCnt := ParameterCnt - 1;
// Create log entry for LimitValues.J6LowerLimit
CreateLogMessagePara1 ( Timestamp   := AxesGroup.State.SystemTime,
                        MessageType := MessageType.CMD,
                        Severity    := Severity.DEBUG,
                        MessageCode := 0,
                        MessageText := 'Command.LimitValues.J6LowerLimit = {1}',
                        Para1       :=  REAL_TO_STRING(_command.LimitValues.J6LowerLimit));


// Return if no parameter is remaining...
IF ( ParameterCnt = 0 ) THEN RETURN; END_IF
// dec remaining parameter(s)                        
ParameterCnt := ParameterCnt - 1;
// Create log entry for LimitValues.E1LowerLimit
CreateLogMessagePara1 ( Timestamp   := AxesGroup.State.SystemTime,
                        MessageType := MessageType.CMD,
                        Severity    := Severity.DEBUG,
                        MessageCode := 0,
                        MessageText := 'Command.LimitValues.E1LowerLimit = {1}',
                        Para1       :=  REAL_TO_STRING(_command.LimitValues.E1LowerLimit));


// Return if no parameter is remaining...
IF ( ParameterCnt = 0 ) THEN RETURN; END_IF
// dec remaining parameter(s)                        
ParameterCnt := ParameterCnt - 1;
// Create log entry for LimitValues.J1UpperLimit
CreateLogMessagePara1 ( Timestamp   := AxesGroup.State.SystemTime,
                        MessageType := MessageType.CMD,
                        Severity    := Severity.DEBUG,
                        MessageCode := 0,
                        MessageText := 'Command.LimitValues.J1UpperLimit = {1}',
                        Para1       :=  REAL_TO_STRING(_command.LimitValues.J1UpperLimit));


// Return if no parameter is remaining...
IF ( ParameterCnt = 0 ) THEN RETURN; END_IF
// dec remaining parameter(s)                        
ParameterCnt := ParameterCnt - 1;
// Create log entry for LimitValues.J2UpperLimit
CreateLogMessagePara1 ( Timestamp   := AxesGroup.State.SystemTime,
                        MessageType := MessageType.CMD,
                        Severity    := Severity.DEBUG,
                        MessageCode := 0,
                        MessageText := 'Command.LimitValues.J2UpperLimit = {1}',
                        Para1       :=  REAL_TO_STRING(_command.LimitValues.J2UpperLimit));


// Return if no parameter is remaining...
IF ( ParameterCnt = 0 ) THEN RETURN; END_IF
// dec remaining parameter(s)                        
ParameterCnt := ParameterCnt - 1;
// Create log entry for LimitValues.J3UpperLimit
CreateLogMessagePara1 ( Timestamp   := AxesGroup.State.SystemTime,
                        MessageType := MessageType.CMD,
                        Severity    := Severity.DEBUG,
                        MessageCode := 0,
                        MessageText := 'Command.LimitValues.J3UpperLimit = {1}',
                        Para1       :=  REAL_TO_STRING(_command.LimitValues.J3UpperLimit));


// Return if no parameter is remaining...
IF ( ParameterCnt = 0 ) THEN RETURN; END_IF
// dec remaining parameter(s)                        
ParameterCnt := ParameterCnt - 1;
// Create log entry for LimitValues.J4UpperLimit
CreateLogMessagePara1 ( Timestamp   := AxesGroup.State.SystemTime,
                        MessageType := MessageType.CMD,
                        Severity    := Severity.DEBUG,
                        MessageCode := 0,
                        MessageText := 'Command.LimitValues.J4UpperLimit = {1}',
                        Para1       :=  REAL_TO_STRING(_command.LimitValues.J4UpperLimit));


// Return if no parameter is remaining...
IF ( ParameterCnt = 0 ) THEN RETURN; END_IF
// dec remaining parameter(s)                        
ParameterCnt := ParameterCnt - 1;
// Create log entry for LimitValues.J5UpperLimit
CreateLogMessagePara1 ( Timestamp   := AxesGroup.State.SystemTime,
                        MessageType := MessageType.CMD,
                        Severity    := Severity.DEBUG,
                        MessageCode := 0,
                        MessageText := 'Command.LimitValues.J5UpperLimit = {1}',
                        Para1       :=  REAL_TO_STRING(_command.LimitValues.J5UpperLimit));


// Return if no parameter is remaining...
IF ( ParameterCnt = 0 ) THEN RETURN; END_IF
// dec remaining parameter(s)                        
ParameterCnt := ParameterCnt - 1;
// Create log entry for LimitValues.J6UpperLimit
CreateLogMessagePara1 ( Timestamp   := AxesGroup.State.SystemTime,
                        MessageType := MessageType.CMD,
                        Severity    := Severity.DEBUG,
                        MessageCode := 0,
                        MessageText := 'Command.LimitValues.J6UpperLimit = {1}',
                        Para1       :=  REAL_TO_STRING(_command.LimitValues.J6UpperLimit));


// Return if no parameter is remaining...
IF ( ParameterCnt = 0 ) THEN RETURN; END_IF
// dec remaining parameter(s)                        
ParameterCnt := ParameterCnt - 1;
// Create log entry for LimitValues.E1UpperLimit
CreateLogMessagePara1 ( Timestamp   := AxesGroup.State.SystemTime,
                        MessageType := MessageType.CMD,
                        Severity    := Severity.DEBUG,
                        MessageCode := 0,
                        MessageText := 'Command.LimitValues.E1UpperLimit = {1}',
                        Para1       :=  REAL_TO_STRING(_command.LimitValues.E1UpperLimit));


// Return if no parameter is remaining...
IF ( ParameterCnt = 0 ) THEN RETURN; END_IF
// dec remaining parameter(s)                        
ParameterCnt := ParameterCnt - 1;
// Create log entry for LimitValues.E2LowerLimit
CreateLogMessagePara1 ( Timestamp   := AxesGroup.State.SystemTime,
                        MessageType := MessageType.CMD,
                        Severity    := Severity.DEBUG,
                        MessageCode := 0,
                        MessageText := 'Command.LimitValues.E2LowerLimit = {1}',
                        Para1       :=  REAL_TO_STRING(_command.LimitValues.E2LowerLimit));


// Return if no parameter is remaining...
IF ( ParameterCnt = 0 ) THEN RETURN; END_IF
// dec remaining parameter(s)                        
ParameterCnt := ParameterCnt - 1;
// Create log entry for LimitValues.E3LowerLimit
CreateLogMessagePara1 ( Timestamp   := AxesGroup.State.SystemTime,
                        MessageType := MessageType.CMD,
                        Severity    := Severity.DEBUG,
                        MessageCode := 0,
                        MessageText := 'Command.LimitValues.E3LowerLimit = {1}',
                        Para1       :=  REAL_TO_STRING(_command.LimitValues.E3LowerLimit));


// Return if no parameter is remaining...
IF ( ParameterCnt = 0 ) THEN RETURN; END_IF
// dec remaining parameter(s)                        
ParameterCnt := ParameterCnt - 1;
// Create log entry for LimitValues.E4LowerLimit
CreateLogMessagePara1 ( Timestamp   := AxesGroup.State.SystemTime,
                        MessageType := MessageType.CMD,
                        Severity    := Severity.DEBUG,
                        MessageCode := 0,
                        MessageText := 'Command.LimitValues.E4LowerLimit = {1}',
                        Para1       :=  REAL_TO_STRING(_command.LimitValues.E4LowerLimit));


